KUKA KRL program: MyProgram_074().src

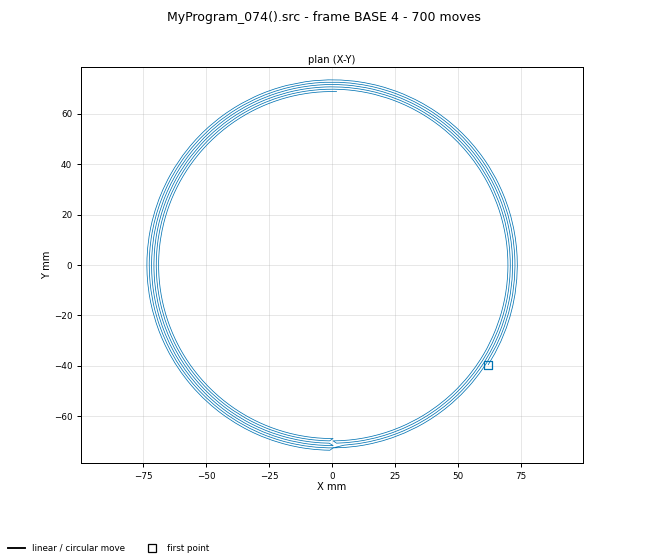
[picture p0: tool path of MyProgram_074().src in frame BASE 4, 700 of 700 moves have a stored position in this frame; points joined in program order, loops and branches not executed]
&ACCESS RVP
&REL 1
&PARAM TEMPLATE = C:\KRC\Roboter\Template\vorgabe
&PARAM EDITMASK = *
DEF MyProgram_074()
; ---- Setting reference (Base) ----
$BASE = BASE_DATA[4]

; --------------------------
; ---- Setting tool (TCP) ----
$TOOL = TOOL_DATA[3]
; --------------------------

$VEL.CP = VEL_APROX_PRINT
Startdeposition()
$VEL.CP = VEL_PRINT
LIN {X 62.0149,Y -39.5352,Z 78,A -36.8264,B 24.9007,C -2.3005,E1 25.1365,E2 121.1791} C_DIS
LIN {X 64.5776,Y -35.1935,Z 78,A -33.5799,B 24.9015,C -2.2916,E1 25.141,E2 117.9704} C_DIS
LIN {X 67.0266,Y -30.2699,Z 78,A -29.6894,B 24.9014,C -2.2926,E1 25.1458,E2 114.0982} C_DIS
LIN {X 69.1793,Y -24.9624,Z 78,A -24.6932,B 24.8988,C -2.3219,E1 25.151,E2 109.0606} C_DIS
LIN {X 70.6037,Y -20.5927,Z 78,A -21.3241,B 24.8984,C -2.3267,E1 25.1538,E2 105.6993} C_DIS
LIN {X 71.7542,Y -16.1353,Z 78,A -17.1231,B 24.8958,C -2.3562,E1 25.1566,E2 101.4529} C_DIS
LIN {X 72.6519,Y -11.4261,Z 78,A -13.91,B 24.8962,C -2.3525,E1 25.1581,E2 98.2674} C_DIS
LIN {X 73.337,Y -5.5339,Z 78,A -9.6921,B 24.8959,C -2.3552,E1 25.1594,E2 94.0681} C_DIS
LIN {X 73.5444,Y -0.3114,Z 78,A -5.4364,B 24.8943,C -2.3735,E1 25.1598,E2 89.7944} C_DIS
LIN {X 73.4622,Y 3.4708,Z 78,A -2.3202,B 24.893,C -2.3879,E1 25.1595,E2 86.6628} C_DIS
LIN {X 73.24,Y 6.6845,Z 78,A 0.445,B 24.8916,C -2.4034,E1 25.1589,E2 83.8775} C_DIS
LIN {X 72.7679,Y 10.6663,Z 78,A 3.6105,B 24.8906,C -2.4143,E1 25.1577,E2 80.7048} C_DIS
LIN {X 72.0794,Y 14.6088,Z 78,A 6.5507,B 24.8902,C -2.4187,E1 25.1561,E2 77.7715} C_DIS
LIN {X 70.9838,Y 19.2388,Z 78,A 9.4181,B 24.8914,C -2.4052,E1 25.1543,E2 74.9524} C_DIS
LIN {X 69.9868,Y 22.5982,Z 78,A 13.0379,B 24.8883,C -2.4394,E1 25.1513,E2 71.2724} C_DIS
LIN {X 68.5839,Y 26.5557,Z 78,A 15.7831,B 24.8889,C -2.4335,E1 25.1486,E2 68.5566} C_DIS
LIN {X 67.3749,Y 29.4866,Z 78,A 19.0656,B 24.886,C -2.4644,E1 25.145,E2 65.2191} C_DIS
LIN {X 65.998,Y 32.4522,Z 78,A 20.5878,B 24.8881,C -2.4414,E1 25.1432,E2 63.7593} C_DIS
LIN {X 64.9381,Y 34.5246,Z 78,A 22.9314,B 24.8863,C -2.4618,E1 25.1401,E2 61.38} C_DIS
LIN {X 62.4288,Y 38.8777,Z 78,A 26.5828,B 24.886,C -2.4644,E1 25.135,E2 57.7411} C_DIS
LIN {X 61.0309,Y 41.038,Z 78,A 29.3198,B 24.8836,C -2.4907,E1 25.1306,E2 54.9554} C_DIS
LIN {X 59.0987,Y 43.7747,Z 78,A 31.7272,B 24.8836,C -2.4912,E1 25.1266,E2 52.5586} C_DIS
LIN {X 56.5702,Y 46.9962,Z 78,A 34.4398,B 24.8841,C -2.4849,E1 25.1219,E2 49.8734} C_DIS
LIN {X 54.0669,Y 49.8561,Z 78,A 37.654,B 24.8828,C -2.4987,E1 25.1159,E2 46.6408} C_DIS
LIN {X 51.7673,Y 52.2397,Z 78,A 39.8636,B 24.8833,C -2.4936,E1 25.1116,E2 44.4527} C_DIS
LIN {X 49.0295,Y 54.8173,Z 78,A 43.1232,B 24.8819,C -2.5088,E1 25.1048,E2 41.1703} C_DIS
LIN {X 46.0603,Y 57.3357,Z 78,A 45.6068,B 24.8828,C -2.499,E1 25.0996,E2 38.7194} C_DIS
LIN {X 42.3941,Y 60.0976,Z 78,A 49.5839,B 24.8811,C -2.5164,E1 25.0906,E2 34.7154} C_DIS
LIN {X 39.5989,Y 61.974,Z 78,A 52.4619,B 24.8801,C -2.5276,E1 25.0838,E2 31.8202} C_DIS
LIN {X 35.9228,Y 64.1746,Z 78,A 55.5006,B 24.8804,C -2.524,E1 25.0765,E2 28.7992} C_DIS
LIN {X 32.8974,Y 65.7773,Z 78,A 58.0417,B 24.8804,C -2.524,E1 25.0702,E2 26.2653} C_DIS
LIN {X 28.2288,Y 67.9124,Z 78,A 62.274,B 24.8794,C -2.5347,E1 25.0594,E2 22.0179} C_DIS
LIN {X 25.5373,Y 68.9696,Z 78,A 64.6555,B 24.8789,C -2.5403,E1 25.0531,E2 19.6282} C_DIS
LIN {X 20.7617,Y 70.5536,Z 78,A 68.6434,B 24.8784,C -2.5451,E1 25.0425,E2 15.6362} C_DIS
LIN {X 17.3304,Y 71.4737,Z 78,A 71.462,B 24.8781,C -2.548,E1 25.0348,E2 12.8146} C_DIS
LIN {X 12.8619,Y 72.4115,Z 78,A 75.4013,B 24.877,C -2.5596,E1 25.0239,E2 8.8522} C_DIS
LIN {X 8.9262,Y 73.002,Z 78,A 77.3268,B 24.8799,C -2.5292,E1 25.0188,E2 7.0007} C_DIS
LIN {X 3.4859,Y 73.4628,Z 78,A 82.4313,B 24.8778,C -2.5516,E1 25.0045,E2 1.8454} C_DIS
LIN {X -1.5466,Y 73.5287,Z 78,A 86.1691,B 24.8783,C -2.5459,E1 24.9941,E2 -1.8791} C_DIS
LIN {X -7.4487,Y 73.1668,Z 78,A 91.0301,B 24.8779,C -2.5504,E1 24.9805,E2 -6.7528} C_DIS
LIN {X -10.6837,Y 72.7654,Z 78,A 93.4689,B 24.8783,C -2.5462,E1 24.9738,E2 -9.1836} C_DIS
LIN {X -17.9304,Y 71.3266,Z 78,A 98.5002,B 24.8805,C -2.5229,E1 24.9602,E2 -14.1655} C_DIS
LIN {X -19.7523,Y 70.8433,Z 78,A 100.539,B 24.8793,C -2.5356,E1 24.9546,E2 -16.238} C_DIS
LIN {X -22.8143,Y 69.9169,Z 78,A 103.3619,B 24.8788,C -2.5411,E1 24.9471,E2 -19.0788} C_DIS
LIN {X -25.9829,Y 68.802,Z 78,A 105.0367,B 24.8813,C -2.5143,E1 24.9428,E2 -20.6933} C_DIS
LIN {X -28.9327,Y 67.6153,Z 78,A 107.5191,B 24.8817,C -2.511,E1 24.9364,E2 -23.1734} C_DIS
LIN {X -30.8582,Y 66.758,Z 78,A 109.859,B 24.8803,C -2.5257,E1 24.9304,E2 -25.5541} C_DIS
LIN {X -35.9812,Y 64.142,Z 78,A 113.8595,B 24.8821,C -2.5064,E1 24.9206,E2 -29.5198} C_DIS
LIN {X -38.9619,Y 62.3763,Z 78,A 116.7798,B 24.8821,C -2.5069,E1 24.9136,E2 -32.4504} C_DIS
LIN {X -42.2245,Y 60.2162,Z 78,A 120.0318,B 24.8821,C -2.5059,E1 24.9061,E2 -35.7108} C_DIS
LIN {X -44.9358,Y 58.2203,Z 78,A 122.322,B 24.8834,C -2.4925,E1 24.901,E2 -37.9773} C_DIS
LIN {X -48.9728,Y 54.868,Z 78,A 127.1321,B 24.8826,C -2.5007,E1 24.8908,E2 -42.8257} C_DIS
LIN {X -51.4287,Y 52.5733,Z 78,A 129.2512,B 24.8843,C -2.4826,E1 24.8866,E2 -44.9105} C_DIS
LIN {X -54.0846,Y 49.8368,Z 78,A 132.8002,B 24.8837,C -2.4891,E1 24.8798,E2 -48.4904} C_DIS
LIN {X -56.3937,Y 47.2085,Z 78,A 135.9816,B 24.8833,C -2.493,E1 24.874,E2 -51.6958} C_DIS
LIN {X -59.2678,Y 43.5445,Z 78,A 138.2236,B 24.8873,C -2.4506,E1 24.8704,E2 -53.8474} C_DIS
LIN {X -62.5156,Y 38.7388,Z 78,A 142.4263,B 24.8891,C -2.4308,E1 24.8639,E2 -58.0238} C_DIS
LIN {X -64.2155,Y 35.8496,Z 78,A 145.4875,B 24.8888,C -2.4337,E1 24.8596,E2 -61.1079} C_DIS
LIN {X -65.2844,Y 33.867,Z 78,A 147.6608,B 24.8884,C -2.4383,E1 24.8567,E2 -63.3037} C_DIS
LIN {X -67.216,Y 29.8477,Z 78,A 150.7781,B 24.8901,C -2.4198,E1 24.8531,E2 -66.3937} C_DIS
LIN {X -68.7386,Y 26.1504,Z 78,A 154.2674,B 24.8901,C -2.419,E1 24.8495,E2 -69.9007} C_DIS
LIN {X -70.2736,Y 21.6899,Z 78,A 157.5058,B 24.8921,C -2.3977,E1 24.8466,E2 -73.1066} C_DIS
LIN {X -71.416,Y 17.5671,Z 78,A 160.9656,B 24.8928,C -2.3902,E1 24.8441,E2 -76.5686} C_DIS
LIN {X -72.0851,Y 14.5798,Z 78,A 163.5914,B 24.893,C -2.3882,E1 24.8426,E2 -79.2052} C_DIS
LIN {X -72.6593,Y 11.3786,Z 78,A 167.1865,B 24.8915,C -2.4048,E1 24.841,E2 -82.8613} C_DIS
LIN {X -73.2264,Y 6.8359,Z 78,A 169.709,B 24.8947,C -2.3692,E1 24.8403,E2 -85.314} C_DIS
LIN {X -73.4955,Y 2.7241,Z 78,A 172.9366,B 24.8955,C -2.3594,E1 24.8398,E2 -88.5374} C_DIS
LIN {X -73.5433,Y -0.4685,Z 78,A 176.0317,B 24.895,C -2.3656,E1 24.8398,E2 -91.6659} C_DIS
LIN {X -73.4495,Y -3.7539,Z 78,A 178.0186,B 24.8969,C -2.3442,E1 24.8401,E2 -93.6137} C_DIS
LIN {X -73.185,Y -7.2754,Z 78,A -179.5399,B 24.8983,C -2.3284,E1 24.8407,E2 -96.0323} C_DIS
LIN {X -72.628,Y -11.5765,Z 78,A -175.831,B 24.8985,C -2.3255,E1 24.8421,E2 -99.7563} C_DIS
LIN {X -72.0901,Y -14.5557,Z 78,A -173.34,B 24.8989,C -2.3213,E1 24.8434,E2 -102.252} C_DIS
LIN {X -71.3296,Y -17.9187,Z 78,A -170.224,B 24.8987,C -2.3232,E1 24.8455,E2 -105.3907} C_DIS
LIN {X -69.8642,Y -22.977,Z 78,A -166.6369,B 24.9008,C -2.2989,E1 24.8484,E2 -108.9406} C_DIS
LIN {X -68.6959,Y -26.2625,Z 78,A -163.9305,B 24.9015,C -2.2908,E1 24.851,E2 -111.6429} C_DIS
LIN {X -67.5462,Y -29.0931,Z 78,A -161.4211,B 24.9019,C -2.2871,E1 24.8537,E2 -114.1572} C_DIS
LIN {X -66.2626,Y -31.9076,Z 78,A -159.1939,B 24.9028,C -2.2761,E1 24.8563,E2 -116.3703} C_DIS
LIN {X -64.5816,Y -35.1861,Z 78,A -155.7371,B 24.9023,C -2.2822,E1 24.8609,E2 -119.8601} C_DIS
LIN {X -62.3685,Y -38.9743,Z 78,A -152.1844,B 24.9028,C -2.2765,E1 24.8661,E2 -123.4176} C_DIS
LIN {X -59.9501,Y -42.6008,Z 78,A -148.9097,B 24.9037,C -2.2652,E1 24.8713,E2 -126.6813} C_DIS
LIN {X -57.585,Y -45.7474,Z 78,A -146.2138,B 24.9051,C -2.249,E1 24.8759,E2 -129.3513} C_DIS
LIN {X -55.9426,Y -47.7416,Z 78,A -144.1882,B 24.9055,C -2.2447,E1 24.8795,E2 -131.376} C_DIS
LIN {X -54.4689,Y -49.4179,Z 78,A -142.4514,B 24.9058,C -2.2408,E1 24.8828,E2 -133.1111} C_DIS
LIN {X -51.2843,Y -52.7143,Z 78,A -138.5837,B 24.9058,C -2.2405,E1 24.8904,E2 -136.9947} C_DIS
LIN {X -47.9483,Y -55.7664,Z 78,A -135.6851,B 24.9077,C -2.2184,E1 24.8963,E2 -139.8522} C_DIS
LIN {X -44.9917,Y -58.1772,Z 78,A -132.2305,B 24.9071,C -2.2249,E1 24.9039,E2 -143.335} C_DIS
LIN {X -42.2829,Y -60.1758,Z 78,A -129.3799,B 24.9071,C -2.2262,E1 24.9104,E2 -146.1986} C_DIS
LIN {X -38.3696,Y -62.7427,Z 78,A -125.7958,B 24.9076,C -2.2191,E1 24.9189,E2 -149.7773} C_DIS
LIN {X -34.6931,Y -64.849,Z 78,A -121.9218,B 24.9068,C -2.2293,E1 24.9285,E2 -153.6865} C_DIS
LIN {X -31.2662,Y -66.5681,Z 78,A -119.5584,B 24.9084,C -2.2099,E1 24.9343,E2 -156.0098} C_DIS
LIN {X -28.0543,Y -67.9846,Z 78,A -116.8143,B 24.9086,C -2.2073,E1 24.9414,E2 -158.7541} C_DIS
LIN {X -23.7093,Y -69.6185,Z 78,A -112.9079,B 24.9082,C -2.2117,E1 24.9517,E2 -162.6787} C_DIS
LIN {X -19.5219,Y -70.9064,Z 78,A -109.3766,B 24.9082,C -2.2126,E1 24.9612,E2 -166.2177} C_DIS
LIN {X -16.3801,Y -71.6976,Z 78,A -107.7838,B 24.9103,C -2.187,E1 24.9654,E2 -167.7519} C_DIS
LIN {X -12.9712,Y -72.3918,Z 78,A -105.3498,B 24.911,C -2.1788,E1 24.972,E2 -170.169} C_DIS
LIN {X -10.941,Y -72.727,Z 78,A -102.2703,B 24.9078,C -2.2172,E1 24.9808,E2 -173.3425} C_DIS
LIN {X -7.0298,Y -73.2084,Z 78,A -100.245,B 24.9101,C -2.1891,E1 24.9862,E2 -175.3022} C_DIS
LIN {X -3.0309,Y -73.4824,Z 78,A -97.4489,B 24.9108,C -2.1806,E1 24.994,E2 -178.079} C_DIS
LIN {X -0.903,Y -73.5406,Z 78,A -94.0962,B 24.907,C -2.2264,E1 25.0036,E2 -181.5406} C_DIS
LIN {X -0.903,Y -73.5406,Z 78,A -94.0962,B 24.907,C -2.2264,E1 25.0036,E2 -181.5406} C_DIS
Enddeposition()
LIN {X 0.4401,Y -72.5902,Z 78,A -93.7193,B 24.9072,C -2.2247,E1 25.0047,E2 -181.9133} C_DIS
Startdeposition()
$VEL.CP = VEL_PRINT
LIN {X -1.5403,Y -72.5975,Z 78,A -97.2134,B 24.9114,C -2.1733,E1 24.9946,E2 -178.2974} C_DIS
LIN {X -6.3605,Y -72.3352,Z 78,A -102.0186,B 24.9134,C -2.1483,E1 24.981,E2 -173.4305} C_DIS
LIN {X -11.1322,Y -71.7552,Z 78,A -104.0226,B 24.9097,C -2.1942,E1 24.9758,E2 -171.5341} C_DIS
LIN {X -15.5858,Y -70.9213,Z 78,A -107.7338,B 24.9099,C -2.192,E1 24.9656,E2 -167.8137} C_DIS
LIN {X -19.0944,Y -70.0583,Z 78,A -111.0187,B 24.9106,C -2.1826,E1 24.9566,E2 -164.5018} C_DIS
LIN {X -21.8748,Y -69.2399,Z 78,A -113.5308,B 24.911,C -2.1787,E1 24.9498,E2 -161.9761} C_DIS
LIN {X -25.901,Y -67.8374,Z 78,A -116.8325,B 24.9106,C -2.1832,E1 24.9412,E2 -158.6783} C_DIS
LIN {X -28.4017,Y -66.8291,Z 78,A -119.2336,B 24.911,C -2.1787,E1 24.935,E2 -156.261} C_DIS
LIN {X -32.57,Y -64.8993,Z 78,A -122.8507,B 24.9106,C -2.1831,E1 24.9259,E2 -152.6452} C_DIS
LIN {X -37.5446,Y -62.1544,Z 78,A -127.452,B 24.9103,C -2.1865,E1 24.9147,E2 -148.0383} C_DIS
LIN {X -41.535,Y -59.5616,Z 78,A -130.5191,B 24.9085,C -2.2089,E1 24.9077,E2 -145.0143} C_DIS
LIN {X -44.3548,Y -57.4925,Z 78,A -133.5609,B 24.9086,C -2.2069,E1 24.9009,E2 -141.957} C_DIS
LIN {X -46.925,Y -55.415,Z 78,A -135.6957,B 24.9073,C -2.2229,E1 24.8963,E2 -139.8522} C_DIS
LIN {X -50.093,Y -52.5699,Z 78,A -140.3066,B 24.9092,C -2.2003,E1 24.8867,E2 -135.1687} C_DIS
LIN {X -52.715,Y -49.9393,Z 78,A -142.4082,B 24.9071,C -2.2258,E1 24.8828,E2 -133.1187} C_DIS
LIN {X -55.1223,Y -47.2686,Z 78,A -145.38,B 24.9068,C -2.229,E1 24.8773,E2 -130.1412} C_DIS
LIN {X -57.2915,Y -44.6156,Z 78,A -147.6991,B 24.9055,C -2.2442,E1 24.8733,E2 -127.8475} C_DIS
LIN {X -59.5737,Y -41.5176,Z 78,A -150.8597,B 24.9051,C -2.2487,E1 24.8681,E2 -124.6824} C_DIS
LIN {X -61.8421,Y -38.0586,Z 78,A -154.1792,B 24.9045,C -2.2557,E1 24.863,E2 -121.3629} C_DIS
LIN {X -63.9816,Y -34.3371,Z 78,A -157.9635,B 24.9045,C -2.2557,E1 24.8578,E2 -117.5587} C_DIS
LIN {X -65.6101,Y -31.1157,Z 78,A -161.4614,B 24.9051,C -2.2491,E1 24.8536,E2 -114.026} C_DIS
LIN {X -67.1485,Y -27.6387,Z 78,A -164.6161,B 24.9047,C -2.2542,E1 24.8502,E2 -110.866} C_DIS
LIN {X -68.6294,Y -23.7246,Z 78,A -166.7374,B 24.9016,C -2.2901,E1 24.8483,E2 -108.8184} C_DIS
LIN {X -69.2974,Y -21.6921,Z 78,A -169.606,B 24.9034,C -2.2689,E1 24.8459,E2 -105.8827} C_DIS
LIN {X -70.4208,Y -17.714,Z 78,A -171.9981,B 24.9009,C -2.2979,E1 24.8442,E2 -103.5458} C_DIS
LIN {X -70.9767,Y -15.3319,Z 78,A -174.239,B 24.901,C -2.2969,E1 24.8429,E2 -101.2895} C_DIS
LIN {X -71.9087,Y -10.0935,Z 78,A -178.0344,B 24.8991,C -2.3188,E1 24.8412,E2 -97.5238} C_DIS
LIN {X -72.2407,Y -7.352,Z 78,A 179.9213,B 24.8983,C -2.3286,E1 24.8405,E2 -95.4907} C_DIS
LIN {X -72.5297,Y -3.511,Z 78,A 176.2296,B 24.8987,C -2.3238,E1 24.8399,E2 -91.7652} C_DIS
LIN {X -72.611,Y 0.6577,Z 78,A 173.3066,B 24.8971,C -2.3423,E1 24.8399,E2 -88.8689} C_DIS
LIN {X -72.5207,Y 3.6858,Z 78,A 171.2509,B 24.8957,C -2.3573,E1 24.84,E2 -86.8366} C_DIS
LIN {X -72.2735,Y 7.0282,Z 78,A 167.488,B 24.8972,C -2.3411,E1 24.841,E2 -83.0126} C_DIS
LIN {X -71.8395,Y 10.581,Z 78,A 165.357,B 24.895,C -2.3652,E1 24.8418,E2 -80.9264} C_DIS
LIN {X -71.4317,Y 13.0495,Z 78,A 162.9633,B 24.8953,C -2.3623,E1 24.843,E2 -78.5114} C_DIS
LIN {X -70.7012,Y 16.5566,Z 78,A 159.5591,B 24.8956,C -2.3586,E1 24.8452,E2 -75.0784} C_DIS
LIN {X -69.6173,Y 20.6438,Z 78,A 157.5721,B 24.892,C -2.3985,E1 24.8466,E2 -73.1753} C_DIS
LIN {X -68.4133,Y 24.3394,Z 78,A 153.7756,B 24.8926,C -2.3918,E1 24.85,E2 -69.3411} C_DIS
LIN {X -66.9712,Y 28.0645,Z 78,A 151.1206,B 24.8908,C -2.4123,E1 24.8527,E2 -66.7202} C_DIS
LIN {X -65.3212,Y 31.7169,Z 78,A 147.7001,B 24.8905,C -2.4159,E1 24.8568,E2 -63.2896} C_DIS
LIN {X -63.8021,Y 34.6702,Z 78,A 145.108,B 24.8897,C -2.4241,E1 24.8601,E2 -60.7035} C_DIS
LIN {X -61.8525,Y 38.0413,Z 78,A 141.0659,B 24.8909,C -2.4113,E1 24.866,E2 -56.61} C_DIS
LIN {X -59.6134,Y 41.4605,Z 78,A 138.9818,B 24.8878,C -2.4455,E1 24.8692,E2 -54.5972} C_DIS
LIN {X -58.5543,Y 42.9433,Z 78,A 136.1975,B 24.8902,C -2.4194,E1 24.874,E2 -51.737} C_DIS
LIN {X -55.7144,Y 46.5691,Z 78,A 133.3525,B 24.8877,C -2.4462,E1 24.8789,E2 -48.943} C_DIS
LIN {X -52.5449,Y 50.1189,Z 78,A 129.9963,B 24.886,C -2.4645,E1 24.8852,E2 -45.6157} C_DIS
LIN {X -48.35,Y 54.1759,Z 78,A 124.8913,B 24.886,C -2.4638,E1 24.8956,E2 -40.488} C_DIS
LIN {X -44.2936,Y 57.5396,Z 78,A 120.5645,B 24.8856,C -2.4689,E1 24.9051,E2 -36.1572} C_DIS
LIN {X -39.9033,Y 60.6668,Z 78,A 116.8787,B 24.8836,C -2.4903,E1 24.9134,E2 -32.51} C_DIS
LIN {X -37.3511,Y 62.2709,Z 78,A 114.5657,B 24.883,C -2.4962,E1 24.9189,E2 -30.2037} C_DIS
LIN {X -35.3335,Y 63.4373,Z 78,A 112.286,B 24.8837,C -2.4891,E1 24.9245,E2 -27.9004} C_DIS
LIN {X -30.6059,Y 65.8484,Z 78,A 108.9963,B 24.8811,C -2.517,E1 24.9326,E2 -24.6684} C_DIS
LIN {X -26.6576,Y 67.5434,Z 78,A 105.0286,B 24.8819,C -2.5079,E1 24.9429,E2 -20.6701} C_DIS
LIN {X -22.7333,Y 68.9644,Z 78,A 101.938,B 24.8811,C -2.5169,E1 24.951,E2 -17.5947} C_DIS
LIN {X -18.8094,Y 70.1353,Z 78,A 98.6328,B 24.8809,C -2.5185,E1 24.9599,E2 -14.288} C_DIS
LIN {X -14.7924,Y 71.0912,Z 78,A 95.2009,B 24.8811,C -2.5172,E1 24.9692,E2 -10.8486} C_DIS
LIN {X -10.3563,Y 71.8714,Z 78,A 91.266,B 24.8817,C -2.5104,E1 24.9801,E2 -6.8938} C_DIS
LIN {X -6.6457,Y 72.3088,Z 78,A 87.8411,B 24.8827,C -2.5002,E1 24.9897,E2 -3.4429} C_DIS
LIN {X -2.8742,Y 72.5571,Z 78,A 85.6748,B 24.8807,C -2.5214,E1 24.9956,E2 -1.3264} C_DIS
LIN {X 2.7685,Y 72.5613,Z 78,A 81.5646,B 24.8798,C -2.5307,E1 25.007,E2 2.7613} C_DIS
LIN {X 7.1833,Y 72.2584,Z 78,A 77.8819,B 24.8803,C -2.5257,E1 25.0173,E2 6.4542} C_DIS
LIN {X 12.2744,Y 71.5691,Z 78,A 73.9452,B 24.8801,C -2.5277,E1 25.0282,E2 10.3828} C_DIS
LIN {X 15.8244,Y 70.8692,Z 78,A 70.7772,B 24.881,C -2.5183,E1 25.0369,E2 13.569} C_DIS
LIN {X 18.9884,Y 70.0869,Z 78,A 68.0915,B 24.8814,C -2.5138,E1 25.0441,E2 16.2612} C_DIS
LIN {X 22.9158,Y 68.9035,Z 78,A 64.8524,B 24.8816,C -2.5113,E1 25.0528,E2 19.5004} C_DIS
LIN {X 25.3422,Y 68.049,Z 78,A 62.5806,B 24.8824,C -2.5031,E1 25.0588,E2 21.7868} C_DIS
LIN {X 29.5259,Y 66.3391,Z 78,A 59.0606,B 24.8826,C -2.5005,E1 25.0678,E2 25.3046} C_DIS
LIN {X 32.6326,Y 64.8693,Z 78,A 56.3222,B 24.883,C -2.4964,E1 25.0746,E2 28.0453} C_DIS
LIN {X 37.1431,Y 62.3953,Z 78,A 52.5098,B 24.883,C -2.4973,E1 25.0839,E2 31.8441} C_DIS
LIN {X 39.8844,Y 60.6793,Z 78,A 49.8553,B 24.8836,C -2.4906,E1 25.0901,E2 34.5059} C_DIS
LIN {X 43.8644,Y 57.8683,Z 78,A 46.2697,B 24.8836,C -2.4911,E1 25.0982,E2 38.0778} C_DIS
LIN {X 46.424,Y 55.8349,Z 78,A 43.4145,B 24.8847,C -2.4788,E1 25.1044,E2 40.9511} C_DIS
LIN {X 49.9897,Y 52.6671,Z 78,A 40.0556,B 24.8843,C -2.4824,E1 25.1113,E2 44.288} C_DIS
LIN {X 52.0972,Y 50.5834,Z 78,A 36.7563,B 24.8872,C -2.4511,E1 25.1178,E2 47.6472} C_DIS
LIN {X 54.8193,Y 47.6195,Z 78,A 34.4891,B 24.8856,C -2.4689,E1 25.1219,E2 49.8621} C_DIS
LIN {X 56.7747,Y 45.271,Z 78,A 31.6954,B 24.8871,C -2.4527,E1 25.1269,E2 52.6812} C_DIS
LIN {X 59.7464,Y 41.2692,Z 78,A 28.2101,B 24.8868,C -2.4555,E1 25.1325,E2 56.143} C_DIS
LIN {X 61.4607,Y 38.67,Z 78,A 24.6138,B 24.8903,C -2.4175,E1 25.138,E2 59.811} C_DIS
LIN {X 63.8046,Y 34.6657,Z 78,A 22.0991,B 24.8883,C -2.4397,E1 25.1413,E2 62.2601} C_DIS
LIN {X 65.6837,Y 30.9582,Z 78,A 18.7462,B 24.8893,C -2.4286,E1 25.1454,E2 65.6214} C_DIS
LIN {X 67.5155,Y 26.7288,Z 78,A 15.5727,B 24.8891,C -2.4314,E1 25.1489,E2 68.7709} C_DIS
LIN {X 68.2892,Y 24.6853,Z 78,A 13.2462,B 24.8911,C -2.4092,E1 25.1511,E2 71.1367} C_DIS
LIN {X 69.7825,Y 20.0803,Z 78,A 9.7819,B 24.8911,C -2.408,E1 25.154,E2 74.5842} C_DIS
LIN {X 71.1056,Y 14.722,Z 78,A 5.4941,B 24.8922,C -2.3967,E1 25.1568,E2 78.8739} C_DIS
LIN {X 71.9388,Y 9.8818,Z 78,A 1.0849,B 24.8947,C -2.3694,E1 25.1587,E2 83.3217} C_DIS
LIN {X 72.4268,Y 5.2153,Z 78,A -2.0955,B 24.8944,C -2.3727,E1 25.1595,E2 86.4755} C_DIS
LIN {X 72.5861,Y 2.009,Z 78,A -4.6685,B 24.8952,C -2.3635,E1 25.1598,E2 89.0548} C_DIS
LIN {X 72.6114,Y -0.594,Z 78,A -6.9772,B 24.8964,C -2.3497,E1 25.1598,E2 91.3824} C_DIS
LIN {X 72.4059,Y -5.4963,Z 78,A -11.0013,B 24.8979,C -2.333,E1 25.1591,E2 95.4219} C_DIS
LIN {X 71.7497,Y -11.1679,Z 78,A -14.7551,B 24.8972,C -2.3403,E1 25.1577,E2 99.1365} C_DIS
LIN {X 71.4279,Y -13.0697,Z 78,A -17.0569,B 24.8996,C -2.3131,E1 25.1566,E2 101.489} C_DIS
LIN {X 70.1423,Y -18.7835,Z 78,A -21.0411,B 24.8993,C -2.3168,E1 25.154,E2 105.4413} C_DIS
LIN {X 68.4563,Y -24.2177,Z 78,A -25.2646,B 24.8998,C -2.3106,E1 25.1504,E2 109.6555} C_DIS
LIN {X 67.1016,Y -27.7519,Z 78,A -28.6725,B 24.9017,C -2.2894,E1 25.1469,E2 113.0946} C_DIS
LIN {X 65.1265,Y -32.1138,Z 78,A -32.6589,B 24.9031,C -2.2723,E1 25.1421,E2 117.1} C_DIS
LIN {X 61.5029,Y -38.6025,Z 78,A -37.7524,B 24.9027,C -2.2775,E1 25.1351,E2 122.1548} C_DIS
LIN {X 59.8419,Y -41.1303,Z 78,A -40.4332,B 24.904,C -2.2625,E1 25.1309,E2 124.8577} C_DIS
LIN {X 58.2027,Y -43.4193,Z 78,A -42.8532,B 24.905,C -2.2509,E1 25.1269,E2 127.2935} C_DIS
LIN {X 55.5723,Y -46.7395,Z 78,A -45.8602,B 24.9049,C -2.2516,E1 25.1216,E2 130.2848} C_DIS
LIN {X 54.2613,Y -48.2546,Z 78,A -47.9078,B 24.9063,C -2.2345,E1 25.1178,E2 132.3638} C_DIS
LIN {X 51.1951,Y -51.4961,Z 78,A -51.2602,B 24.9067,C -2.2306,E1 25.1113,E2 135.7108} C_DIS
LIN {X 47.6851,Y -54.762,Z 78,A -54.8564,B 24.907,C -2.2271,E1 25.1038,E2 139.3009} C_DIS
LIN {X 44.6981,Y -57.2264,Z 78,A -58.062,B 24.9079,C -2.2163,E1 25.0968,E2 142.52} C_DIS
LIN {X 41.9624,Y -59.2618,Z 78,A -60.5827,B 24.9079,C -2.2155,E1 25.0912,E2 145.0336} C_DIS
LIN {X 39.158,Y -61.1506,Z 78,A -62.9782,B 24.9077,C -2.2179,E1 25.0856,E2 147.4156} C_DIS
LIN {X 36.3366,Y -62.8683,Z 78,A -66.0755,B 24.9092,C -2.1996,E1 25.0781,E2 150.5466} C_DIS
LIN {X 33.766,Y -64.2853,Z 78,A -68.5201,B 24.9099,C -2.1922,E1 25.072,E2 153.0018} C_DIS
LIN {X 28.7007,Y -66.7017,Z 78,A -72.6086,B 24.9097,C -2.1946,E1 25.0617,E2 157.0743} C_DIS
LIN {X 23.8439,Y -68.5875,Z 78,A -76.9358,B 24.9106,C -2.1834,E1 25.0503,E2 161.419} C_DIS
LIN {X 20.0624,Y -69.7876,Z 78,A -79.3866,B 24.9094,C -2.198,E1 25.0439,E2 163.8307} C_DIS
LIN {X 15.8946,Y -70.8531,Z 78,A -82.834,B 24.9098,C -2.1932,E1 25.0346,E2 167.2843} C_DIS
LIN {X 12.6894,Y -71.4964,Z 78,A -85.9596,B 24.9111,C -2.1766,E1 25.0259,E2 170.4457} C_DIS
LIN {X 9.7952,Y -71.9511,Z 78,A -88.3417,B 24.9114,C -2.1732,E1 25.0193,E2 172.8339} C_DIS
LIN {X 5.0583,Y -72.4374,Z 78,A -91.4313,B 24.9101,C -2.1887,E1 25.0108,E2 175.8847} C_DIS
LIN {X 0.4401,Y -72.5902,Z 78,A -93.7169,B 24.9072,C -2.2237,E1 25.0047,E2 178.0866} C_DIS
Enddeposition()
LIN {X 0.4401,Y -72.5902,Z 78,A -93.7169,B 24.9072,C -2.2237,E1 25.0047,E2 178.0866} C_DIS
Startdeposition()
$VEL.CP = VEL_PRINT
LIN {X 4.7456,Y -71.5252,Z 78,A -90.38,B 24.9061,C -2.2377,E1 25.014,E2 174.7179} C_DIS
LIN {X 10.2822,Y -70.9414,Z 78,A -86.6436,B 24.9074,C -2.2214,E1 25.0243,E2 171.0228} C_DIS
LIN {X 14.8753,Y -70.1232,Z 78,A -82.6289,B 24.9065,C -2.232,E1 25.0354,E2 166.9876} C_DIS
LIN {X 19.1531,Y -69.0775,Z 78,A -79.4537,B 24.907,C -2.2263,E1 25.0439,E2 163.8307} C_DIS
LIN {X 22.1838,Y -68.1635,Z 78,A -76.5584,B 24.9059,C -2.2391,E1 25.0517,E2 160.9103} C_DIS
LIN {X 25.58,Y -66.9633,Z 78,A -73.669,B 24.9056,C -2.2432,E1 25.0593,E2 158.0173} C_DIS
LIN {X 28.1777,Y -65.913,Z 78,A -70.7706,B 24.9038,C -2.2645,E1 25.0668,E2 155.0752} C_DIS
LIN {X 31.4442,Y -64.4179,Z 78,A -68.6285,B 24.9051,C -2.2489,E1 25.0721,E2 152.9757} C_DIS
LIN {X 34.006,Y -63.1031,Z 78,A -65.4024,B 24.9026,C -2.2786,E1 25.0802,E2 149.6887} C_DIS
LIN {X 37.6579,Y -60.9951,Z 78,A -63.3344,B 24.9052,C -2.2484,E1 25.085,E2 147.6984} C_DIS
LIN {X 40.9313,Y -58.8473,Z 78,A -59.8082,B 24.9037,C -2.2656,E1 25.0932,E2 144.1434} C_DIS
LIN {X 44.6413,Y -56.0849,Z 78,A -55.918,B 24.9026,C -2.2788,E1 25.1018,E2 140.2362} C_DIS
LIN {X 46.9592,Y -54.1597,Z 78,A -53.8364,B 24.9029,C -2.275,E1 25.1062,E2 138.1717} C_DIS
LIN {X 49.4403,Y -51.9046,Z 78,A -51.189,B 24.9024,C -2.2803,E1 25.1116,E2 135.5226} C_DIS
LIN {X 51.6215,Y -49.7352,Z 78,A -48.6933,B 24.9018,C -2.2873,E1 25.1165,E2 133.0209} C_DIS
LIN {X 54.1776,Y -46.9387,Z 78,A -45.9867,B 24.902,C -2.2858,E1 25.1216,E2 130.33} C_DIS
LIN {X 55.8769,Y -44.9022,Z 78,A -43.2005,B 24.8999,C -2.3103,E1 25.1265,E2 127.4988} C_DIS
LIN {X 58.5293,Y -41.3847,Z 78,A -39.4132,B 24.8984,C -2.3275,E1 25.1328,E2 123.6891} C_DIS
LIN {X 60.4416,Y -38.5387,Z 78,A -37.643,B 24.9001,C -2.3072,E1 25.1354,E2 121.9756} C_DIS
LIN {X 62.7833,Y -34.5948,Z 78,A -34.0069,B 24.8993,C -2.3168,E1 25.1405,E2 118.3358} C_DIS
LIN {X 64.3772,Y -31.5262,Z 78,A -30.4988,B 24.8967,C -2.3464,E1 25.145,E2 114.7764} C_DIS
LIN {X 66.0027,Y -27.9648,Z 78,A -27.8624,B 24.8971,C -2.3415,E1 25.1479,E2 112.1659} C_DIS
LIN {X 67.4223,Y -24.3447,Z 78,A -24.9219,B 24.8967,C -2.3461,E1 25.1508,E2 109.2309} C_DIS
LIN {X 68.732,Y -20.3541,Z 78,A -21.6942,B 24.8961,C -2.3527,E1 25.1535,E2 106.0058} C_DIS
LIN {X 69.3673,Y -18.0723,Z 78,A -19.3717,B 24.8945,C -2.3711,E1 25.1552,E2 103.6533} C_DIS
LIN {X 70.2697,Y -14.1634,Z 78,A -16.1801,B 24.8936,C -2.3807,E1 25.1571,E2 100.4575} C_DIS
LIN {X 70.8276,Y -11.0375,Z 78,A -13.4231,B 24.8923,C -2.3952,E1 25.1583,E2 97.6827} C_DIS
LIN {X 71.4579,Y -5.6701,Z 78,A -10.2024,B 24.894,C -2.3771,E1 25.1593,E2 94.5237} C_DIS
LIN {X 71.6804,Y -0.5619,Z 78,A -5.9042,B 24.8923,C -2.3961,E1 25.1598,E2 90.2062} C_DIS
LIN {X 71.6628,Y 1.7243,Z 78,A -3.383,B 24.8899,C -2.4219,E1 25.1596,E2 87.639} C_DIS
LIN {X 71.4672,Y 5.5535,Z 78,A -0.6145,B 24.8899,C -2.423,E1 25.1591,E2 84.8843} C_DIS
LIN {X 71.0755,Y 9.3088,Z 78,A 2.2221,B 24.8894,C -2.4272,E1 25.1582,E2 82.0545} C_DIS
LIN {X 70.4749,Y 13.1001,Z 78,A 5.3987,B 24.8883,C -2.4398,E1 25.1568,E2 78.8668} C_DIS
LIN {X 69.846,Y 16.1216,Z 78,A 7.8978,B 24.8875,C -2.4483,E1 25.1552,E2 76.3622} C_DIS
LIN {X 69.2762,Y 18.4189,Z 78,A 9.6227,B 24.8875,C -2.4492,E1 25.154,E2 74.6451} C_DIS
LIN {X 68.5086,Y 21.0943,Z 78,A 12.6696,B 24.8846,C -2.4795,E1 25.1515,E2 71.5439} C_DIS
LIN {X 67.3709,Y 24.4855,Z 78,A 14.6422,B 24.8862,C -2.4624,E1 25.1497,E2 69.6229} C_DIS
LIN {X 66.078,Y 27.7861,Z 78,A 17.4411,B 24.8855,C -2.4695,E1 25.1468,E2 66.8227} C_DIS
LIN {X 64.7824,Y 30.6838,Z 78,A 20.3834,B 24.8838,C -2.4882,E1 25.1433,E2 63.8521} C_DIS
LIN {X 63.3875,Y 33.4724,Z 78,A 23.0827,B 24.8826,C -2.5008,E1 25.1398,E2 61.1372} C_DIS
LIN {X 60.4909,Y 38.4619,Z 78,A 27.1516,B 24.8829,C -2.4974,E1 25.134,E2 57.097} C_DIS
LIN {X 58.0066,Y 42.1153,Z 78,A 30.7393,B 24.882,C -2.5078,E1 25.1282,E2 53.5025} C_DIS
LIN {X 56.4708,Y 44.1539,Z 78,A 32.7586,B 24.8815,C -2.5121,E1 25.1248,E2 51.4826} C_DIS
LIN {X 54.3523,Y 46.7365,Z 78,A 35.3621,B 24.8811,C -2.5163,E1 25.1201,E2 48.8809} C_DIS
LIN {X 52.248,Y 49.0767,Z 78,A 38.0654,B 24.8801,C -2.5271,E1 25.115,E2 46.164} C_DIS
LIN {X 50.0307,Y 51.3367,Z 78,A 40.8868,B 24.8788,C -2.5404,E1 25.1093,E2 43.3229} C_DIS
LIN {X 46.6072,Y 54.4626,Z 78,A 44.0428,B 24.8796,C -2.5325,E1 25.1028,E2 40.1982} C_DIS
LIN {X 44.1184,Y 56.4988,Z 78,A 46.7,B 24.8789,C -2.5395,E1 25.097,E2 37.5343} C_DIS
LIN {X 41.3446,Y 58.5587,Z 78,A 49.8804,B 24.8774,C -2.5557,E1 25.0897,E2 34.3268} C_DIS
LIN {X 38.4968,Y 60.4685,Z 78,A 52.2029,B 24.8781,C -2.5485,E1 25.0843,E2 32.0288} C_DIS
LIN {X 34.7944,Y 62.6718,Z 78,A 55.9316,B 24.8769,C -2.5611,E1 25.0752,E2 28.2815} C_DIS
LIN {X 31.8195,Y 64.2331,Z 78,A 58.1051,B 24.8779,C -2.5507,E1 25.0699,E2 26.1385} C_DIS
LIN {X 27.457,Y 66.2168,Z 78,A 62.7104,B 24.8755,C -2.5755,E1 25.058,E2 21.4856} C_DIS
LIN {X 24.3786,Y 67.4099,Z 78,A 64.7509,B 24.8768,C -2.562,E1 25.0527,E2 19.4813} C_DIS
LIN {X 19.894,Y 68.8673,Z 78,A 68.8778,B 24.8756,C -2.5742,E1 25.0416,E2 15.3328} C_DIS
LIN {X 16.207,Y 69.8263,Z 78,A 71.4099,B 24.8767,C -2.5626,E1 25.0349,E2 12.8321} C_DIS
LIN {X 13.3918,Y 70.4206,Z 78,A 73.889,B 24.8762,C -2.5682,E1 25.028,E2 10.3427} C_DIS
LIN {X 8.4945,Y 71.1775,Z 78,A 77.6599,B 24.8766,C -2.5643,E1 25.0177,E2 6.5844} C_DIS
LIN {X 5.6815,Y 71.4569,Z 78,A 80.1178,B 24.876,C -2.5696,E1 25.0108,E2 4.1154} C_DIS
LIN {X 2.0734,Y 71.6526,Z 78,A 83.3877,B 24.8751,C -2.5791,E1 25.0016,E2 0.8237} C_DIS
LIN {X -2.6527,Y 71.6346,Z 78,A 86.6386,B 24.8765,C -2.5648,E1 24.9926,E2 -2.3934} C_DIS
LIN {X -5.5367,Y 71.4685,Z 78,A 89.261,B 24.8758,C -2.5716,E1 24.9853,E2 -5.0332} C_DIS
LIN {X -8.5001,Y 71.1769,Z 78,A 92.1858,B 24.8747,C -2.5839,E1 24.9771,E2 -7.9891} C_DIS
LIN {X -12.2549,Y 70.6285,Z 78,A 94.2077,B 24.8773,C -2.5567,E1 24.9717,E2 -9.9481} C_DIS
LIN {X -14.8215,Y 70.1346,Z 78,A 96.5057,B 24.877,C -2.5601,E1 24.9654,E2 -12.2569} C_DIS
LIN {X -17.8595,Y 69.422,Z 78,A 99.8666,B 24.8751,C -2.579,E1 24.9561,E2 -15.6676} C_DIS
LIN {X -21.6353,Y 68.3408,Z 78,A 101.9911,B 24.8779,C -2.5507,E1 24.9506,E2 -17.7284} C_DIS
LIN {X -24.561,Y 67.3434,Z 78,A 104.8128,B 24.8773,C -2.5561,E1 24.9431,E2 -20.5685} C_DIS
LIN {X -28.6535,Y 65.7065,Z 78,A 108.1234,B 24.8783,C -2.5461,E1 24.9347,E2 -23.8627} C_DIS
LIN {X -31.4543,Y 64.4141,Z 78,A 110.6726,B 24.8785,C -2.5443,E1 24.9282,E2 -26.4141} C_DIS
LIN {X -34.6857,Y 62.7325,Z 78,A 113.5777,B 24.879,C -2.5393,E1 24.9211,E2 -29.3155} C_DIS
LIN {X -37.5827,Y 61.0405,Z 78,A 115.996,B 24.88,C -2.5283,E1 24.9153,E2 -31.715} C_DIS
LIN {X -39.265,Y 59.9724,Z 78,A 117.9079,B 24.8796,C -2.5327,E1 24.9108,E2 -33.6436} C_DIS
LIN {X -42.1667,Y 57.9683,Z 78,A 120.7317,B 24.8801,C -2.5272,E1 24.9044,E2 -36.4641} C_DIS
LIN {X -44.6227,Y 56.1002,Z 78,A 124.0535,B 24.8787,C -2.542,E1 24.897,E2 -39.8334} C_DIS
LIN {X -47.6444,Y 53.5577,Z 78,A 125.9008,B 24.8823,C -2.5046,E1 24.8933,E2 -41.5988} C_DIS
LIN {X -50.9656,Y 50.4071,Z 78,A 129.8828,B 24.8823,C -2.5034,E1 24.8853,E2 -45.5944} C_DIS
LIN {X -55.0352,Y 45.9296,Z 78,A 135.6083,B 24.8816,C -2.5116,E1 24.8746,E2 -51.3653} C_DIS
LIN {X -57.2232,Y 43.1729,Z 78,A 137.8458,B 24.8835,C -2.491,E1 24.8709,E2 -53.5642} C_DIS
LIN {X -59.979,Y 39.2549,Z 78,A 141.8221,B 24.8842,C -2.4839,E1 24.8646,E2 -57.5432} C_DIS
LIN {X -61.8182,Y 36.289,Z 78,A 144.8547,B 24.8844,C -2.4815,E1 24.8603,E2 -60.5858} C_DIS
LIN {X -63.9731,Y 32.3399,Z 78,A 148.8046,B 24.8846,C -2.479,E1 24.8552,E2 -64.551} C_DIS
LIN {X -65.5804,Y 28.9428,Z 78,A 150.9695,B 24.8872,C -2.4512,E1 24.8528,E2 -66.6612} C_DIS
LIN {X -66.7013,Y 26.2546,Z 78,A 153.3809,B 24.8877,C -2.446,E1 24.8503,E2 -69.0738} C_DIS
LIN {X -68.5791,Y 20.8668,Z 78,A 157.6371,B 24.8896,C -2.4252,E1 24.8465,E2 -73.3045} C_DIS
LIN {X -69.6392,Y 16.9928,Z 78,A 161.01,B 24.8902,C -2.4188,E1 24.8441,E2 -76.6817} C_DIS
LIN {X -70.4464,Y 13.257,Z 78,A 164.0995,B 24.891,C -2.4099,E1 24.8423,E2 -79.7683} C_DIS
LIN {X -70.8079,Y 11.165,Z 78,A 165.8492,B 24.8914,C -2.4058,E1 24.8415,E2 -81.5183} C_DIS
LIN {X -71.3182,Y 7.221,Z 78,A 169.5456,B 24.8913,C -2.4072,E1 24.8403,E2 -85.2403} C_DIS
LIN {X -71.612,Y 3.1786,Z 78,A 172.3552,B 24.8931,C -2.3873,E1 24.8399,E2 -88.0193} C_DIS
LIN {X -71.6827,Y 0.204,Z 78,A 174.8132,B 24.8936,C -2.3815,E1 24.8398,E2 -90.4783} C_DIS
LIN {X -71.6082,Y -3.2677,Z 78,A 177.8285,B 24.8939,C -2.3781,E1 24.8401,E2 -93.5036} C_DIS
LIN {X -71.4035,Y -6.3233,Z 78,A -179.9861,B 24.8951,C -2.3646,E1 24.8406,E2 -95.6697} C_DIS
LIN {X -71.0987,Y -9.13,Z 78,A -177.7635,B 24.8958,C -2.3568,E1 24.8413,E2 -97.887} C_DIS
LIN {X -70.5626,Y -12.6212,Z 78,A -174.6844,B 24.896,C -2.3537,E1 24.8427,E2 -100.9772} C_DIS
LIN {X -69.8932,Y -15.9174,Z 78,A -172.0856,B 24.8969,C -2.3435,E1 24.8442,E2 -103.5669} C_DIS
LIN {X -68.8202,Y -20.0566,Z 78,A -168.2294,B 24.8969,C -2.3431,E1 24.8471,E2 -107.4446} C_DIS
LIN {X -67.5155,Y -24.0838,Z 78,A -165.0727,B 24.8983,C -2.3281,E1 24.8499,E2 -110.5832} C_DIS
LIN {X -66.1112,Y -27.7073,Z 78,A -161.6303,B 24.8984,C -2.3269,E1 24.8536,E2 -114.042} C_DIS
LIN {X -64.4509,Y -31.3782,Z 78,A -158.8586,B 24.9001,C -2.3077,E1 24.8569,E2 -116.7829} C_DIS
LIN {X -62.196,Y -35.6376,Z 78,A -154.9613,B 24.9009,C -2.2984,E1 24.8621,E2 -120.6785} C_DIS
LIN {X -60.3641,Y -38.6595,Z 78,A -152.1132,B 24.9015,C -2.2916,E1 24.8663,E2 -123.525} C_DIS
LIN {X -58.521,Y -41.3974,Z 78,A -149.2156,B 24.9015,C -2.2911,E1 24.8709,E2 -126.4356} C_DIS
LIN {X -56.0963,Y -44.6277,Z 78,A -146.3014,B 24.9028,C -2.2761,E1 24.8758,E2 -129.3279} C_DIS
LIN {X -54.1771,Y -46.9392,Z 78,A -144.007,B 24.9035,C -2.2681,E1 24.8799,E2 -131.6139} C_DIS
LIN {X -52.6697,Y -48.6243,Z 78,A -142.3153,B 24.9041,C -2.2615,E1 24.8831,E2 -133.2972} C_DIS
LIN {X -50.3477,Y -51.0243,Z 78,A -139.4767,B 24.9041,C -2.2598,E1 24.8887,E2 -136.144} C_DIS
LIN {X -48.774,Y -52.5313,Z 78,A -137.1048,B 24.9032,C -2.2713,E1 24.8936,E2 -138.5528} C_DIS
LIN {X -45.9571,Y -55.0123,Z 78,A -134.6135,B 24.9047,C -2.2534,E1 24.8988,E2 -141.0113} C_DIS
LIN {X -43.4522,Y -57.0125,Z 78,A -132.2937,B 24.9056,C -2.2431,E1 24.9039,E2 -143.315} C_DIS
LIN {X -41.1732,Y -58.6791,Z 78,A -129.6931,B 24.9052,C -2.2476,E1 24.9098,E2 -145.9353} C_DIS
LIN {X -38.006,Y -60.7776,Z 78,A -126.5556,B 24.9054,C -2.2454,E1 24.9172,E2 -149.0777} C_DIS
LIN {X -34.6164,Y -62.7712,Z 78,A -123.7077,B 24.9064,C -2.2338,E1 24.9241,E2 -151.9065} C_DIS
LIN {X -32.1972,Y -64.0458,Z 78,A -121.1625,B 24.9059,C -2.2399,E1 24.9304,E2 -154.473} C_DIS
LIN {X -27.4604,Y -66.2153,Z 78,A -117.5139,B 24.9073,C -2.2227,E1 24.9397,E2 -158.0894} C_DIS
LIN {X -22.8339,Y -67.9482,Z 78,A -112.864,B 24.9062,C -2.2367,E1 24.952,E2 -162.782} C_DIS
LIN {X -19.0389,Y -69.1088,Z 78,A -110.1004,B 24.9072,C -2.2243,E1 24.9593,E2 -165.5206} C_DIS
LIN {X -16.472,Y -69.7651,Z 78,A -107.8925,B 24.9071,C -2.2254,E1 24.9653,E2 -167.7344} C_DIS
LIN {X -11.4509,Y -70.7629,Z 78,A -104.1134,B 24.9079,C -2.216,E1 24.9757,E2 -171.495} C_DIS
LIN {X -9.3461,Y -71.0707,Z 78,A -101.6475,B 24.9063,C -2.2353,E1 24.9826,E2 -174.0086} C_DIS
LIN {X -5.4444,Y -71.4756,Z 78,A -98.2206,B 24.9056,C -2.2428,E1 24.9922,E2 -177.4549} C_DIS
LIN {X -1.7879,Y -71.6613,Z 78,A -96.3463,B 24.9079,C -2.2157,E1 24.9973,E2 -179.2652} C_DIS
LIN {X 0.4083,Y -71.6761,Z 78,A -93.3356,B 24.9051,C -2.2492,E1 25.0059,E2 -182.355} C_DIS
Enddeposition()
LIN {X 0.4083,Y -71.6761,Z 78,A -93.3356,B 24.9051,C -2.2492,E1 25.0059,E2 -182.355} C_DIS
Startdeposition()
$VEL.CP = VEL_PRINT
LIN {X -1.1606,Y -70.7419,Z 78,A -96.5417,B 24.908,C -2.2146,E1 24.9967,E2 -179.0671} C_DIS
LIN {X -4.4902,Y -70.6092,Z 78,A -99.78,B 24.9091,C -2.2009,E1 24.9876,E2 -175.7955} C_DIS
LIN {X -8.1917,Y -70.2755,Z 78,A -102.5281,B 24.9086,C -2.2077,E1 24.98,E2 -173.062} C_DIS
LIN {X -11.4245,Y -69.8233,Z 78,A -104.7482,B 24.9077,C -2.2188,E1 24.9739,E2 -170.8663} C_DIS
LIN {X -14.1074,Y -69.3307,Z 78,A -107.6091,B 24.9089,C -2.2037,E1 24.966,E2 -167.9663} C_DIS
LIN {X -17.7821,Y -68.4805,Z 78,A -110.4283,B 24.9083,C -2.211,E1 24.9584,E2 -165.1607} C_DIS
LIN {X -20.2752,Y -67.7841,Z 78,A -113.3487,B 24.9098,C -2.1927,E1 24.9504,E2 -162.1918} C_DIS
LIN {X -23.8184,Y -66.6223,Z 78,A -115.6227,B 24.9081,C -2.2129,E1 24.9445,E2 -159.9615} C_DIS
LIN {X -26.5116,Y -65.5966,Z 78,A -118.5135,B 24.909,C -2.202,E1 24.937,E2 -157.0384} C_DIS
LIN {X -29.4785,Y -64.319,Z 78,A -120.6091,B 24.9078,C -2.2171,E1 24.9317,E2 -154.9735} C_DIS
LIN {X -32.5367,Y -62.8272,Z 78,A -123.3291,B 24.9074,C -2.2213,E1 24.9249,E2 -152.2564} C_DIS
LIN {X -34.4089,Y -61.8206,Z 78,A -125.9359,B 24.909,C -2.2031,E1 24.9185,E2 -149.5986} C_DIS
LIN {X -37.8203,Y -59.7937,Z 78,A -128.3959,B 24.9071,C -2.2252,E1 24.9127,E2 -147.1836} C_DIS
LIN {X -40.3209,Y -58.1376,Z 78,A -130.4397,B 24.906,C -2.238,E1 24.9081,E2 -145.1635} C_DIS
LIN {X -42.4139,Y -56.6288,Z 78,A -132.6511,B 24.906,C -2.2387,E1 24.9031,E2 -142.9459} C_DIS
LIN {X -44.6556,Y -54.8785,Z 78,A -135.0271,B 24.9058,C -2.2412,E1 24.8979,E2 -140.5669} C_DIS
LIN {X -47.4249,Y -52.5039,Z 78,A -138.1042,B 24.9055,C -2.2441,E1 24.8914,E2 -137.4846} C_DIS
LIN {X -50.7718,Y -49.2746,Z 78,A -141.7987,B 24.9047,C -2.2535,E1 24.8841,E2 -133.797} C_DIS
LIN {X -53.2293,Y -46.6089,Z 78,A -144.796,B 24.9043,C -2.2586,E1 24.8785,E2 -130.7986} C_DIS
LIN {X -55.2392,Y -44.2105,Z 78,A -147.3517,B 24.9038,C -2.264,E1 24.8739,E2 -128.2438} C_DIS
LIN {X -56.5343,Y -42.5397,Z 78,A -149.0373,B 24.9034,C -2.2687,E1 24.8711,E2 -126.5613} C_DIS
LIN {X -58.8656,Y -39.2518,Z 78,A -152.8262,B 24.9037,C -2.2652,E1 24.8651,E2 -122.7455} C_DIS
LIN {X -60.5416,Y -36.6126,Z 78,A -155.9116,B 24.9042,C -2.2598,E1 24.8606,E2 -119.6312} C_DIS
LIN {X -62.6289,Y -32.9146,Z 78,A -158.356,B 24.9016,C -2.2906,E1 24.8574,E2 -117.2474} C_DIS
LIN {X -63.839,Y -30.5017,Z 78,A -160.311,B 24.9006,C -2.3017,E1 24.8551,E2 -115.3083} C_DIS
LIN {X -65.072,Y -27.7756,Z 78,A -163.9685,B 24.9023,C -2.2818,E1 24.8509,E2 -111.5832} C_DIS
LIN {X -66.5875,Y -23.9161,Z 78,A -166.3386,B 24.8996,C -2.3128,E1 24.8487,E2 -109.2736} C_DIS
LIN {X -67.4472,Y -21.3676,Z 78,A -168.7493,B 24.8996,C -2.3142,E1 24.8466,E2 -106.8525} C_DIS
LIN {X -68.6032,Y -17.3045,Z 78,A -171.9442,B 24.8982,C -2.3293,E1 24.8443,E2 -103.6751} C_DIS
LIN {X -69.2015,Y -14.7317,Z 78,A -174.0163,B 24.8975,C -2.3373,E1 24.843,E2 -101.6098} C_DIS
LIN {X -69.6643,Y -12.3557,Z 78,A -176.0893,B 24.8972,C -2.3409,E1 24.842,E2 -99.5333} C_DIS
LIN {X -70.0788,Y -9.7344,Z 78,A -178.1234,B 24.8964,C -2.35,E1 24.8411,E2 -97.5089} C_DIS
LIN {X -70.4268,Y -6.7738,Z 78,A 179.2036,B 24.8962,C -2.352,E1 24.8403,E2 -94.8246} C_DIS
LIN {X -70.6106,Y -4.4705,Z 78,A 177.4199,B 24.8955,C -2.3598,E1 24.84,E2 -93.0487} C_DIS
LIN {X -70.7317,Y -1.7026,Z 78,A 175.2166,B 24.8948,C -2.3677,E1 24.8398,E2 -90.8512} C_DIS
LIN {X -70.7481,Y 0.7512,Z 78,A 173.033,B 24.8946,C -2.3698,E1 24.8398,E2 -88.6595} C_DIS
LIN {X -70.6154,Y 4.3997,Z 78,A 170.2355,B 24.8935,C -2.3826,E1 24.8402,E2 -85.8757} C_DIS
LIN {X -70.3618,Y 7.414,Z 78,A 167.4581,B 24.8934,C -2.3834,E1 24.8409,E2 -83.0835} C_DIS
LIN {X -69.8297,Y 11.3864,Z 78,A 164.8059,B 24.8913,C -2.4064,E1 24.842,E2 -80.4703} C_DIS
LIN {X -69.4582,Y 13.4651,Z 78,A 162.6406,B 24.8917,C -2.402,E1 24.8431,E2 -78.2818} C_DIS
LIN {X -68.7464,Y 16.7237,Z 78,A 159.9806,B 24.8909,C -2.4114,E1 24.8448,E2 -75.6285} C_DIS
LIN {X -67.7309,Y 20.4548,Z 78,A 156.5158,B 24.8906,C -2.414,E1 24.8474,E2 -72.1499} C_DIS
LIN {X -66.6885,Y 23.6313,Z 78,A 154.1318,B 24.8893,C -2.4292,E1 24.8496,E2 -69.7886} C_DIS
LIN {X -65.6268,Y 26.4374,Z 78,A 151.6539,B 24.8887,C -2.4355,E1 24.8521,E2 -67.3119} C_DIS
LIN {X -64.6057,Y 28.8428,Z 78,A 149.1567,B 24.8888,C -2.4336,E1 24.8549,E2 -64.7965} C_DIS
LIN {X -63.1299,Y 31.9444,Z 78,A 146.992,B 24.8869,C -2.4551,E1 24.8575,E2 -62.6714} C_DIS
LIN {X -61.8519,Y 34.3529,Z 78,A 144.298,B 24.8873,C -2.4509,E1 24.8612,E2 -59.9532} C_DIS
LIN {X -60.3704,Y 36.8943,Z 78,A 141.7167,B 24.887,C -2.4534,E1 24.8649,E2 -57.3644} C_DIS
LIN {X -57.7512,Y 40.8732,Z 78,A 138.3386,B 24.8851,C -2.4743,E1 24.8701,E2 -54.0195} C_DIS
LIN {X -55.8727,Y 43.4058,Z 78,A 135.3118,B 24.8854,C -2.4707,E1 24.8753,E2 -50.9698} C_DIS
LIN {X -52.2066,Y 47.7518,Z 78,A 131.0152,B 24.8837,C -2.4891,E1 24.8831,E2 -46.6976} C_DIS
LIN {X -50.0933,Y 49.9653,Z 78,A 128.7274,B 24.8828,C -2.4993,E1 24.8875,E2 -44.4243} C_DIS
LIN {X -47.0444,Y 52.8452,Z 78,A 124.6178,B 24.8835,C -2.4913,E1 24.8961,E2 -40.279} C_DIS
LIN {X -42.8613,Y 56.2923,Z 78,A 120.6489,B 24.8817,C -2.51,E1 24.9047,E2 -36.3398} C_DIS
LIN {X -40.0786,Y 58.3053,Z 78,A 117.8586,B 24.8812,C -2.5153,E1 24.911,E2 -33.5527} C_DIS
LIN {X -37.8167,Y 59.798,Z 78,A 115.1754,B 24.8819,C -2.5084,E1 24.9174,E2 -30.8445} C_DIS
LIN {X -34.6055,Y 61.7108,Z 78,A 112.6963,B 24.8802,C -2.5261,E1 24.9233,E2 -28.4001} C_DIS
LIN {X -31.9017,Y 63.1517,Z 78,A 110.1261,B 24.88,C -2.5281,E1 24.9297,E2 -25.8278} C_DIS
LIN {X -29.205,Y 64.4425,Z 78,A 107.8617,B 24.8793,C -2.5354,E1 24.9354,E2 -23.575} C_DIS
LIN {X -26.4928,Y 65.6043,Z 78,A 104.8802,B 24.8803,C -2.5251,E1 24.9432,E2 -20.5623} C_DIS
LIN {X -22.5709,Y 67.0545,Z 78,A 102.1233,B 24.8785,C -2.5439,E1 24.9503,E2 -17.8447} C_DIS
LIN {X -17.603,Y 68.5265,Z 78,A 97.9114,B 24.8781,C -2.548,E1 24.9616,E2 -13.6356} C_DIS
LIN {X -14.9565,Y 69.1525,Z 78,A 95.5605,B 24.8783,C -2.5464,E1 24.968,E2 -11.278} C_DIS
LIN {X -12.0251,Y 69.7228,Z 78,A 93.4383,B 24.8774,C -2.5553,E1 24.9738,E2 -9.1747} C_DIS
LIN {X -9.0156,Y 70.1746,Z 78,A 90.8965,B 24.8774,C -2.5551,E1 24.9808,E2 -6.6302} C_DIS
LIN {X -5.4728,Y 70.5395,Z 78,A 87.865,B 24.8776,C -2.5529,E1 24.9893,E2 -3.5921} C_DIS
LIN {X -2.6283,Y 70.7037,Z 78,A 85.4306,B 24.8779,C -2.5506,E1 24.9961,E2 -1.1516} C_DIS
LIN {X -0.6042,Y 70.7489,Z 78,A 83.6463,B 24.8782,C -2.5475,E1 25.0011,E2 0.6401} C_DIS
LIN {X 3.7978,Y 70.6494,Z 78,A 80.2205,B 24.8778,C -2.5512,E1 25.0106,E2 4.0563} C_DIS
LIN {X 6.8563,Y 70.4192,Z 78,A 77.7681,B 24.8778,C -2.5518,E1 25.0174,E2 6.506} C_DIS
LIN {X 10.7839,Y 69.9246,Z 78,A 74.4082,B 24.8782,C -2.5472,E1 25.0268,E2 9.8738} C_DIS
LIN {X 14.0509,Y 69.3423,Z 78,A 71.8923,B 24.8779,C -2.5504,E1 25.0336,E2 12.3792} C_DIS
LIN {X 17.0736,Y 68.661,Z 78,A 69.1817,B 24.8785,C -2.544,E1 25.041,E2 15.1012} C_DIS
LIN {X 20.8216,Y 67.6179,Z 78,A 66.1451,B 24.8785,C -2.5447,E1 25.0491,E2 18.131} C_DIS
LIN {X 23.5359,Y 66.722,Z 78,A 63.075,B 24.8805,C -2.5236,E1 25.0574,E2 21.2449} C_DIS
LIN {X 27.071,Y 65.3689,Z 78,A 60.7822,B 24.8789,C -2.5401,E1 25.0632,E2 23.4933} C_DIS
LIN {X 30.1538,Y 64.0047,Z 78,A 58.1209,B 24.879,C -2.5388,E1 25.0699,E2 26.1511} C_DIS
LIN {X 33.8025,Y 62.1538,Z 78,A 54.1378,B 24.8811,C -2.5172,E1 25.0798,E2 30.1741} C_DIS
LIN {X 36.72,Y 60.4764,Z 78,A 52.1303,B 24.8797,C -2.5318,E1 25.0846,E2 32.1407} C_DIS
LIN {X 40.148,Y 58.2578,Z 78,A 48.8721,B 24.88,C -2.5279,E1 25.0921,E2 35.3976} C_DIS
LIN {X 42.4906,Y 56.5712,Z 78,A 46.476,B 24.8806,C -2.5223,E1 25.0975,E2 37.7983} C_DIS
LIN {X 44.9575,Y 54.6323,Z 78,A 43.9521,B 24.881,C -2.5181,E1 25.103,E2 40.3227} C_DIS
LIN {X 47.1777,Y 52.7258,Z 78,A 41,B 24.8829,C -2.4981,E1 25.1093,E2 43.3104} C_DIS
LIN {X 49.8524,Y 50.2048,Z 78,A 38.2013,B 24.883,C -2.4966,E1 25.1148,E2 46.1009} C_DIS
LIN {X 52.6811,Y 47.2276,Z 78,A 35.348,B 24.8825,C -2.5019,E1 25.1202,E2 48.929} C_DIS
LIN {X 54.6878,Y 44.8907,Z 78,A 32.8756,B 24.883,C -2.4968,E1 25.1246,E2 51.4023} C_DIS
LIN {X 56.4291,Y 42.6797,Z 78,A 30.6893,B 24.8833,C -2.4939,E1 25.1284,E2 53.5851} C_DIS
LIN {X 58.9342,Y 39.148,Z 78,A 27.2475,B 24.8839,C -2.4869,E1 25.1339,E2 57.0265} C_DIS
LIN {X 61.5676,Y 34.8619,Z 78,A 23.0343,B 24.8853,C -2.4724,E1 25.14,E2 61.2524} C_DIS
LIN {X 63.0002,Y 32.1982,Z 78,A 20.6544,B 24.8857,C -2.4677,E1 25.143,E2 63.6309} C_DIS
LIN {X 63.9884,Y 30.1887,Z 78,A 18.7867,B 24.8863,C -2.4612,E1 25.1453,E2 65.504} C_DIS
LIN {X 66.1142,Y 25.1929,Z 78,A 14.6407,B 24.8868,C -2.4556,E1 25.1497,E2 69.6404} C_DIS
LIN {X 67.241,Y 22.0102,Z 78,A 11.7829,B 24.8879,C -2.4441,E1 25.1523,E2 72.5092} C_DIS
LIN {X 68.075,Y 19.2755,Z 78,A 9.4515,B 24.8886,C -2.4368,E1 25.1542,E2 74.8447} C_DIS
LIN {X 68.6971,Y 16.9257,Z 78,A 7.2578,B 24.8897,C -2.4245,E1 25.1557,E2 77.0546} C_DIS
LIN {X 69.6779,Y 12.2799,Z 78,A 3.6332,B 24.8902,C -2.4189,E1 25.1577,E2 80.6714} C_DIS
LIN {X 70.1486,Y 9.2165,Z 78,A 1.4751,B 24.89,C -2.4209,E1 25.1585,E2 82.812} C_DIS
LIN {X 70.5002,Y 5.9652,Z 78,A -1.8039,B 24.8924,C -2.3949,E1 25.1594,E2 86.1329} C_DIS
LIN {X 70.7247,Y 1.9528,Z 78,A -4.6264,B 24.8922,C -2.3967,E1 25.1598,E2 88.9344} C_DIS
LIN {X 70.7487,Y -0.6505,Z 78,A -6.5539,B 24.8923,C -2.3951,E1 25.1598,E2 90.8543} C_DIS
LIN {X 70.6027,Y -4.587,Z 78,A -9.9057,B 24.8937,C -2.3804,E1 25.1594,E2 94.2209} C_DIS
LIN {X 70.1104,Y -9.5111,Z 78,A -14.0328,B 24.8951,C -2.3643,E1 25.1581,E2 98.3616} C_DIS
LIN {X 69.4928,Y -13.2855,Z 78,A -17.4922,B 24.8969,C -2.3444,E1 25.1564,E2 101.8478} C_DIS
LIN {X 68.5894,Y -17.3584,Z 78,A -20.2851,B 24.8964,C -2.3502,E1 25.1546,E2 104.6109} C_DIS
LIN {X 67.7961,Y -20.2348,Z 78,A -22.9393,B 24.8976,C -2.336,E1 25.1525,E2 107.2833} C_DIS
LIN {X 66.831,Y -23.2252,Z 78,A -25.148,B 24.8975,C -2.3376,E1 25.1506,E2 109.4759} C_DIS
LIN {X 65.7743,Y -26.0678,Z 78,A -28.0501,B 24.8992,C -2.3176,E1 25.1476,E2 112.409} C_DIS
LIN {X 63.6333,Y -30.9298,Z 78,A -32.5128,B 24.9007,C -2.3004,E1 25.1424,E2 116.8882} C_DIS
LIN {X 61.5741,Y -34.8502,Z 78,A -35.9773,B 24.9013,C -2.2934,E1 25.1377,E2 120.3513} C_DIS
LIN {X 59.7034,Y -37.9651,Z 78,A -39.6265,B 24.9037,C -2.2657,E1 25.1322,E2 124.0473} C_DIS
LIN {X 57.1986,Y -41.6425,Z 78,A -41.6904,B 24.9009,C -2.2983,E1 25.129,E2 126.0243} C_DIS
LIN {X 56.1943,Y -42.9878,Z 78,A -43.8316,B 24.9031,C -2.2731,E1 25.1253,E2 128.2149} C_DIS
LIN {X 53.5013,Y -46.2975,Z 78,A -47.6049,B 24.9046,C -2.2555,E1 25.1185,E2 132.0125} C_DIS
LIN {X 51.2157,Y -48.8127,Z 78,A -49.7713,B 24.9038,C -2.2647,E1 25.1144,E2 134.1477} C_DIS
LIN {X 48.4274,Y -51.5804,Z 78,A -52.8194,B 24.9041,C -2.2608,E1 25.1082,E2 137.1924} C_DIS
LIN {X 46.1561,Y -53.6236,Z 78,A -54.9359,B 24.9038,C -2.2649,E1 25.1039,E2 139.2907} C_DIS
LIN {X 42.7254,Y -56.3941,Z 78,A -58.6558,B 24.9048,C -2.2531,E1 25.0957,E2 143.0246} C_DIS
LIN {X 41.1953,Y -57.5214,Z 78,A -60.8456,B 24.9065,C -2.2325,E1 25.0907,E2 145.2555} C_DIS
LIN {X 37.8501,Y -59.7771,Z 78,A -63.4669,B 24.9056,C -2.2435,E1 25.0846,E2 147.8422} C_DIS
LIN {X 34.549,Y -61.7423,Z 78,A -66.3651,B 24.9056,C -2.2435,E1 25.0776,E2 150.7312} C_DIS
LIN {X 32.0042,Y -63.0993,Z 78,A -69.1923,B 24.907,C -2.2266,E1 25.0706,E2 153.5909} C_DIS
LIN {X 28.1443,Y -64.9128,Z 78,A -72.2161,B 24.9065,C -2.2327,E1 25.0629,E2 156.5926} C_DIS
LIN {X 23.943,Y -66.5777,Z 78,A -76.2007,B 24.9076,C -2.2191,E1 25.0525,E2 160.6005} C_DIS
LIN {X 20.5613,Y -67.699,Z 78,A -79.0594,B 24.9078,C -2.2164,E1 25.0449,E2 163.4604} C_DIS
LIN {X 17.1157,Y -68.6508,Z 78,A -82.2601,B 24.9088,C -2.2056,E1 25.0362,E2 166.6819} C_DIS
LIN {X 12.9496,Y -69.5575,Z 78,A -85.3532,B 24.9082,C -2.2118,E1 25.0278,E2 169.7564} C_DIS
LIN {X 10.0708,Y -70.031,Z 78,A -87.3052,B 24.9075,C -2.2207,E1 25.0225,E2 171.6854} C_DIS
LIN {X 5.8385,Y -70.5103,Z 78,A -90.9567,B 24.9081,C -2.2136,E1 25.0123,E2 175.3514} C_DIS
LIN {X 1.7707,Y -70.7302,Z 78,A -94.4742,B 24.9086,C -2.2068,E1 25.0024,E2 178.8839} C_DIS
LIN {X 1.7707,Y -70.7302,Z 78,A -94.4742,B 24.9086,C -2.2068,E1 25.0024,E2 178.8839} C_DIS
Enddeposition()
LIN {X 0.3843,Y -69.8184,Z 78,A -94.5954,B 24.9052,C -2.248,E1 25.0024,E2 178.9073} C_DIS
Startdeposition()
$VEL.CP = VEL_PRINT
LIN {X 3.3748,Y -69.7396,Z 78,A -91.878,B 24.9046,C -2.2555,E1 25.01,E2 176.1728} C_DIS
LIN {X 6.7049,Y -69.4981,Z 78,A -89.1101,B 24.9044,C -2.2576,E1 25.0177,E2 173.4015} C_DIS
LIN {X 9.6724,Y -69.1471,Z 78,A -86.8135,B 24.9046,C -2.2551,E1 25.024,E2 171.1125} C_DIS
LIN {X 12.5857,Y -68.6769,Z 78,A -84.2807,B 24.9042,C -2.2599,E1 25.031,E2 168.5712} C_DIS
LIN {X 15.5466,Y -68.0675,Z 78,A -81.5997,B 24.9036,C -2.2673,E1 25.0384,E2 165.876} C_DIS
LIN {X 18.6337,Y -67.289,Z 78,A -79.252,B 24.9039,C -2.2631,E1 25.0447,E2 163.5422} C_DIS
LIN {X 21.3777,Y -66.467,Z 78,A -77.0089,B 24.9039,C -2.2631,E1 25.0506,E2 161.3033} C_DIS
LIN {X 23.9927,Y -65.5684,Z 78,A -74.4278,B 24.903,C -2.2742,E1 25.0575,E2 158.7009} C_DIS
LIN {X 27.0204,Y -64.3798,Z 78,A -72.013,B 24.9032,C -2.2712,E1 25.0637,E2 156.2988} C_DIS
LIN {X 29.6073,Y -63.232,Z 78,A -69.6631,B 24.9029,C -2.2755,E1 25.0697,E2 153.9446} C_DIS
LIN {X 33.9476,Y -61.0117,Z 78,A -65.8375,B 24.9027,C -2.2775,E1 25.0791,E2 150.125} C_DIS
LIN {X 36.1922,Y -59.7075,Z 78,A -63.6812,B 24.9023,C -2.282,E1 25.0843,E2 147.9646} C_DIS
LIN {X 38.5253,Y -58.2295,Z 78,A -60.9021,B 24.9007,C -2.3003,E1 25.0909,E2 145.1514} C_DIS
LIN {X 41.9033,Y -55.8478,Z 78,A -56.966,B 24.8988,C -2.3223,E1 25.0998,E2 141.1773} C_DIS
LIN {X 45.0713,Y -53.3246,Z 78,A -55.0008,B 24.9014,C -2.2922,E1 25.1039,E2 139.2907} C_DIS
LIN {X 47.5445,Y -51.1325,Z 78,A -51.8886,B 24.8999,C -2.3094,E1 25.1104,E2 136.1504} C_DIS
LIN {X 49.6372,Y -49.102,Z 78,A -48.336,B 24.8966,C -2.3475,E1 25.1175,E2 132.5229} C_DIS
LIN {X 52.825,Y -45.6563,Z 78,A -45.9157,B 24.8993,C -2.3172,E1 25.1218,E2 130.185} C_DIS
LIN {X 54.5298,Y -43.6063,Z 78,A -43.2145,B 24.8975,C -2.3372,E1 25.1266,E2 127.449} C_DIS
LIN {X 56.8498,Y -40.5334,Z 78,A -39.542,B 24.8955,C -2.3601,E1 25.1327,E2 123.7401} C_DIS
LIN {X 58.9651,Y -37.3914,Z 78,A -37.3347,B 24.897,C -2.3435,E1 25.136,E2 121.5833} C_DIS
LIN {X 60.3523,Y -35.1083,Z 78,A -35.2183,B 24.8966,C -2.3476,E1 25.139,E2 119.468} C_DIS
LIN {X 61.5421,Y -32.978,Z 78,A -32.5053,B 24.8943,C -2.3734,E1 25.1426,E2 116.7082} C_DIS
LIN {X 63.7708,Y -28.4293,Z 78,A -28.9559,B 24.8947,C -2.3686,E1 25.1468,E2 113.1894} C_DIS
LIN {X 65.006,Y -25.4771,Z 78,A -26.4315,B 24.8943,C -2.3737,E1 25.1494,E2 110.667} C_DIS
LIN {X 66.5642,Y -21.0737,Z 78,A -22.8076,B 24.8937,C -2.3795,E1 25.1527,E2 107.0496} C_DIS
LIN {X 67.2617,Y -18.73,Z 78,A -20.6072,B 24.8927,C -2.3912,E1 25.1544,E2 104.8342} C_DIS
LIN {X 67.9804,Y -15.9236,Z 78,A -18.3035,B 24.8922,C -2.3966,E1 25.1559,E2 102.5311} C_DIS
LIN {X 68.508,Y -13.4756,Z 78,A -16.2943,B 24.8917,C -2.4018,E1 25.1571,E2 100.5213} C_DIS
LIN {X 68.9349,Y -11.091,Z 78,A -14.2595,B 24.8911,C -2.4094,E1 25.158,E2 98.4805} C_DIS
LIN {X 69.3398,Y -8.1759,Z 78,A -11.7107,B 24.89,C -2.4209,E1 25.1589,E2 95.9197} C_DIS
LIN {X 69.6285,Y -5.184,Z 78,A -9.4727,B 24.8899,C -2.4222,E1 25.1594,E2 93.6917} C_DIS
LIN {X 69.7778,Y -2.451,Z 78,A -7.4962,B 24.8899,C -2.4218,E1 25.1597,E2 91.7279} C_DIS
LIN {X 69.8184,Y -0.518,Z 78,A -5.7069,B 24.8889,C -2.4326,E1 25.1597,E2 89.9239} C_DIS
LIN {X 69.7905,Y 2.0383,Z 78,A -3.6143,B 24.8884,C -2.4391,E1 25.1597,E2 87.8284} C_DIS
LIN {X 69.6343,Y 5.1072,Z 78,A -1.033,B 24.8875,C -2.4487,E1 25.1592,E2 85.2397} C_DIS
LIN {X 69.4011,Y 7.6476,Z 78,A 1.2077,B 24.8865,C -2.4594,E1 25.1586,E2 82.987} C_DIS
LIN {X 69.0138,Y 10.5808,Z 78,A 3.3889,B 24.8865,C -2.46,E1 25.1577,E2 80.8172} C_DIS
LIN {X 68.4737,Y 13.6506,Z 78,A 6.0203,B 24.8855,C -2.4699,E1 25.1564,E2 78.1777} C_DIS
LIN {X 67.8254,Y 16.5703,Z 78,A 8.4072,B 24.885,C -2.4755,E1 25.1549,E2 75.7913} C_DIS
LIN {X 67.1263,Y 19.2081,Z 78,A 10.6321,B 24.8844,C -2.4819,E1 25.1532,E2 73.5643} C_DIS
LIN {X 66.3372,Y 21.779,Z 78,A 12.8073,B 24.8839,C -2.4875,E1 25.1514,E2 71.3881} C_DIS
LIN {X 65.4135,Y 24.4141,Z 78,A 15.7662,B 24.8815,C -2.5128,E1 25.1485,E2 68.3859} C_DIS
LIN {X 63.8546,Y 28.2414,Z 78,A 18.3632,B 24.8827,C -2.5003,E1 25.1457,E2 65.8327} C_DIS
LIN {X 62.7092,Y 30.7006,Z 78,A 20.654,B 24.8819,C -2.5083,E1 25.1429,E2 63.5355} C_DIS
LIN {X 61.6592,Y 32.7576,Z 78,A 22.4913,B 24.8816,C -2.5118,E1 25.1405,E2 61.6995} C_DIS
LIN {X 60.5515,Y 34.7617,Z 78,A 24.5463,B 24.8806,C -2.5217,E1 25.1377,E2 59.6318} C_DIS
LIN {X 58.5459,Y 38.0445,Z 78,A 27.3624,B 24.8808,C -2.5205,E1 25.1336,E2 56.8328} C_DIS
LIN {X 56.3866,Y 41.1755,Z 78,A 30.6397,B 24.8796,C -2.5325,E1 25.1283,E2 53.5432} C_DIS
LIN {X 54.5424,Y 43.5904,Z 78,A 33.31,B 24.8786,C -2.5432,E1 25.1237,E2 50.8601} C_DIS
LIN {X 52.341,Y 46.2106,Z 78,A 36.0963,B 24.878,C -2.549,E1 25.1186,E2 48.0727} C_DIS
LIN {X 50.0725,Y 48.6588,Z 78,A 38.807,B 24.8775,C -2.5541,E1 25.1134,E2 45.3616} C_DIS
LIN {X 47.4303,Y 51.2378,Z 78,A 41.8062,B 24.877,C -2.5595,E1 25.1073,E2 42.3621} C_DIS
LIN {X 44.9303,Y 53.4442,Z 78,A 44.4769,B 24.8767,C -2.563,E1 25.1017,E2 39.6936} C_DIS
LIN {X 42.8028,Y 55.1619,Z 78,A 46.8091,B 24.8761,C -2.5694,E1 25.0966,E2 37.3548} C_DIS
LIN {X 40.3363,Y 56.9905,Z 78,A 49.1815,B 24.8761,C -2.5698,E1 25.0912,E2 34.9899} C_DIS
LIN {X 37.9692,Y 58.5943,Z 78,A 51.6603,B 24.8753,C -2.577,E1 25.0854,E2 32.5023} C_DIS
LIN {X 35.1859,Y 60.3051,Z 78,A 55.1636,B 24.8728,C -2.6026,E1 25.0769,E2 28.9489} C_DIS
LIN {X 31.7551,Y 62.181,Z 78,A 57.2859,B 24.8752,C -2.5782,E1 25.0718,E2 26.8904} C_DIS
LIN {X 29.0448,Y 63.4934,Z 78,A 59.994,B 24.8743,C -2.5872,E1 25.0649,E2 24.1679} C_DIS
LIN {X 26.4414,Y 64.6199,Z 78,A 62.0701,B 24.8747,C -2.5832,E1 25.0596,E2 22.1062} C_DIS
LIN {X 23.9912,Y 65.5689,Z 78,A 64.3336,B 24.8743,C -2.588,E1 25.0536,E2 19.8363} C_DIS
LIN {X 21.7706,Y 66.3398,Z 78,A 66.7077,B 24.873,C -2.6009,E1 25.0473,E2 17.436} C_DIS
LIN {X 16.8835,Y 67.749,Z 78,A 70.4425,B 24.8738,C -2.5924,E1 25.0373,E2 13.7274} C_DIS
LIN {X 14.2805,Y 68.3446,Z 78,A 72.6081,B 24.8738,C -2.5928,E1 25.0314,E2 11.5637} C_DIS
LIN {X 11.6341,Y 68.8442,Z 78,A 74.9129,B 24.8735,C -2.596,E1 25.025,E2 9.2537} C_DIS
LIN {X 9.0095,Y 69.2365,Z 78,A 76.9279,B 24.8738,C -2.5925,E1 25.0195,E2 7.2489} C_DIS
LIN {X 6.3854,Y 69.5276,Z 78,A 79.0783,B 24.8738,C -2.5924,E1 25.0135,E2 5.1002} C_DIS
LIN {X 3.7897,Y 69.7173,Z 78,A 81.3177,B 24.8736,C -2.5949,E1 25.0073,E2 2.8556} C_DIS
LIN {X 0.6698,Y 69.8174,Z 78,A 83.9599,B 24.8734,C -2.5966,E1 24.9999,E2 0.2099} C_DIS
LIN {X -2.3359,Y 69.7814,Z 78,A 86.3323,B 24.8737,C -2.5936,E1 24.9933,E2 -2.1557} C_DIS
LIN {X -5.002,Y 69.6414,Z 78,A 88.6034,B 24.8736,C -2.5947,E1 24.9869,E2 -4.4301} C_DIS
LIN {X -8.2866,Y 69.3269,Z 78,A 91.1756,B 24.8741,C -2.59,E1 24.9798,E2 -6.9927} C_DIS
LIN {X -10.861,Y 68.9705,Z 78,A 93.1095,B 24.8747,C -2.5839,E1 24.9745,E2 -8.9136} C_DIS
LIN {X -12.8132,Y 68.6355,Z 78,A 95.0346,B 24.8741,C -2.5898,E1 24.9692,E2 -10.8547} C_DIS
LIN {X -15.4094,Y 68.0992,Z 78,A 97.1854,B 24.8743,C -2.5873,E1 24.9633,E2 -13.0023} C_DIS
LIN {X -17.9584,Y 67.4716,Z 78,A 99.3128,B 24.8746,C -2.5846,E1 24.9576,E2 -15.1263} C_DIS
LIN {X -21.1114,Y 66.5532,Z 78,A 101.822,B 24.8753,C -2.5773,E1 24.9509,E2 -17.6223} C_DIS
LIN {X -23.1316,Y 65.877,Z 78,A 103.9259,B 24.8747,C -2.5835,E1 24.9453,E2 -19.745} C_DIS
LIN {X -26.2423,Y 64.7009,Z 78,A 106.4592,B 24.8755,C -2.5753,E1 24.9387,E2 -22.2642} C_DIS
LIN {X -28.5624,Y 63.7108,Z 78,A 108.5538,B 24.8757,C -2.5728,E1 24.9334,E2 -24.3579} C_DIS
LIN {X -30.8719,Y 62.6243,Z 78,A 110.656,B 24.876,C -2.5698,E1 24.9281,E2 -26.4583} C_DIS
LIN {X -33.0876,Y 61.4827,Z 78,A 112.6989,B 24.8764,C -2.5663,E1 24.9231,E2 -28.4986} C_DIS
LIN {X -35.3544,Y 60.2077,Z 78,A 115.6135,B 24.875,C -2.5805,E1 24.9159,E2 -31.4557} C_DIS
LIN {X -38.0962,Y 58.5124,Z 78,A 118.1826,B 24.8756,C -2.5737,E1 24.9099,E2 -34.017} C_DIS
LIN {X -42.1435,Y 55.6673,Z 78,A 121.7671,B 24.8775,C -2.5547,E1 24.9019,E2 -37.5688} C_DIS
LIN {X -45.0757,Y 53.3208,Z 78,A 124.8345,B 24.8782,C -2.5477,E1 24.8953,E2 -40.631} C_DIS
LIN {X -47.6806,Y 51.0045,Z 78,A 127.4163,B 24.8794,C -2.535,E1 24.89,E2 -43.1929} C_DIS
LIN {X -49.3839,Y 49.3582,Z 78,A 129.644,B 24.8792,C -2.5367,E1 24.8856,E2 -45.434} C_DIS
LIN {X -51.4696,Y 47.1778,Z 78,A 132.0869,B 24.8799,C -2.5299,E1 24.8809,E2 -47.8714} C_DIS
LIN {X -53.6766,Y 44.6506,Z 78,A 134.7524,B 24.8807,C -2.521,E1 24.8761,E2 -50.5278} C_DIS
LIN {X -54.8056,Y 43.2575,Z 78,A 137.2778,B 24.8788,C -2.5405,E1 24.8717,E2 -53.1116} C_DIS
LIN {X -57.1281,Y 40.1417,Z 78,A 139.5734,B 24.8815,C -2.5121,E1 24.868,E2 -55.3507} C_DIS
LIN {X -58.8194,Y 37.6185,Z 78,A 142.056,B 24.8822,C -2.505,E1 24.8642,E2 -57.8288} C_DIS
LIN {X -60.3805,Y 35.0593,Z 78,A 144.5098,B 24.8829,C -2.4979,E1 24.8607,E2 -60.2784} C_DIS
LIN {X -61.7353,Y 32.6131,Z 78,A 147.4458,B 24.8822,C -2.5053,E1 24.8568,E2 -63.2476} C_DIS
LIN {X -63.6295,Y 28.7427,Z 78,A 150.0484,B 24.8851,C -2.4746,E1 24.8538,E2 -65.791} C_DIS
LIN {X -64.4355,Y 26.8884,Z 78,A 152.0571,B 24.8848,C -2.4771,E1 24.8516,E2 -67.8168} C_DIS
LIN {X -65.4373,Y 24.3512,Z 78,A 154.4862,B 24.8851,C -2.4745,E1 24.8491,E2 -70.2532} C_DIS
LIN {X -66.7366,Y 20.521,Z 78,A 157.4659,B 24.8867,C -2.457,E1 24.8466,E2 -73.2081} C_DIS
LIN {X -67.7129,Y 17.0281,Z 78,A 161.109,B 24.8862,C -2.4621,E1 24.8439,E2 -76.8847} C_DIS
LIN {X -68.4692,Y 13.6734,Z 78,A 163.6367,B 24.8876,C -2.4468,E1 24.8425,E2 -79.3909} C_DIS
LIN {X -69.0275,Y 10.4925,Z 78,A 166.181,B 24.8886,C -2.4362,E1 24.8414,E2 -81.9248} C_DIS
LIN {X -69.4054,Y 7.607,Z 78,A 168.4108,B 24.8896,C -2.4252,E1 24.8406,E2 -84.1417} C_DIS
LIN {X -69.6226,Y 5.2582,Z 78,A 170.5809,B 24.8897,C -2.4241,E1 24.8401,E2 -86.3222} C_DIS
LIN {X -69.7838,Y 2.2559,Z 78,A 172.9892,B 24.8905,C -2.415,E1 24.8398,E2 -88.7233} C_DIS
LIN {X -69.8179,Y -0.601,Z 78,A 175.4169,B 24.8911,C -2.4093,E1 24.8398,E2 -91.1522} C_DIS
LIN {X -69.7325,Y -3.5138,Z 78,A 177.7946,B 24.8918,C -2.4015,E1 24.8401,E2 -93.5254} C_DIS
LIN {X -69.5335,Y -6.321,Z 78,A -179.8993,B 24.8924,C -2.3942,E1 24.8406,E2 -95.8278} C_DIS
LIN {X -69.2088,Y -9.2231,Z 78,A -177.4581,B 24.893,C -2.3877,E1 24.8414,E2 -98.2681} C_DIS
LIN {X -68.766,Y -12.0901,Z 78,A -175.1343,B 24.8938,C -2.3791,E1 24.8425,E2 -100.5852} C_DIS
LIN {X -68.2291,Y -14.8207,Z 78,A -172.8151,B 24.8943,C -2.3729,E1 24.8438,E2 -102.9032} C_DIS
LIN {X -67.6945,Y -17.0997,Z 78,A -170.5872,B 24.8943,C -2.3737,E1 24.8453,E2 -105.1462} C_DIS
LIN {X -66.4011,Y -21.5815,Z 78,A -166.9409,B 24.8956,C -2.3584,E1 24.8482,E2 -108.7768} C_DIS
LIN {X -65.3712,Y -24.5256,Z 78,A -164.4282,B 24.8964,C -2.3499,E1 24.8506,E2 -111.2835} C_DIS
LIN {X -64.0279,Y -27.8441,Z 78,A -161.4614,B 24.8971,C -2.3422,E1 24.8538,E2 -114.2484} C_DIS
LIN {X -62.757,Y -30.6036,Z 78,A -158.9358,B 24.8976,C -2.336,E1 24.8568,E2 -116.7729} C_DIS
LIN {X -61.4962,Y -33.0627,Z 78,A -156.3199,B 24.8975,C -2.3376,E1 24.8603,E2 -119.4066} C_DIS
LIN {X -59.5431,Y -36.4627,Z 78,A -153.4777,B 24.8989,C -2.3208,E1 24.8643,E2 -122.2234} C_DIS
LIN {X -57.9911,Y -38.8842,Z 78,A -150.523,B 24.8983,C -2.3282,E1 24.8689,E2 -125.2105} C_DIS
LIN {X -55.933,Y -41.7898,Z 78,A -148.1489,B 24.9,C -2.3087,E1 24.8728,E2 -127.5497} C_DIS
LIN {X -54.152,Y -44.0731,Z 78,A -145.7243,B 24.9004,C -2.3043,E1 24.877,E2 -129.9749} C_DIS
LIN {X -52.2811,Y -46.2785,Z 78,A -143.2118,B 24.9006,C -2.3021,E1 24.8816,E2 -132.4935} C_DIS
LIN {X -50.6431,Y -48.0649,Z 78,A -141.2751,B 24.901,C -2.2966,E1 24.8853,E2 -134.4256} C_DIS
LIN {X -48.0713,Y -50.6371,Z 78,A -137.8312,B 24.9007,C -2.301,E1 24.8922,E2 -137.8945} C_DIS
LIN {X -44.8008,Y -53.5518,Z 78,A -134.7509,B 24.9023,C -2.2823,E1 24.8987,E2 -140.9421} C_DIS
LIN {X -42.2907,Y -55.5565,Z 78,A -132.1496,B 24.9027,C -2.2768,E1 24.9044,E2 -143.5399} C_DIS
LIN {X -39.2424,Y -57.7487,Z 78,A -128.3681,B 24.9018,C -2.2882,E1 24.9131,E2 -147.3614} C_DIS
LIN {X -34.2014,Y -60.87,Z 78,A -124.1814,B 24.9037,C -2.2651,E1 24.9231,E2 -151.5059} C_DIS
LIN {X -31.935,Y -62.089,Z 78,A -122.0693,B 24.904,C -2.2624,E1 24.9283,E2 -153.6175} C_DIS
LIN {X -29.203,Y -63.4202,Z 78,A -119.5738,B 24.9042,C -2.2596,E1 24.9346,E2 -156.1126} C_DIS
LIN {X -26.4273,Y -64.6256,Z 78,A -117.1925,B 24.9046,C -2.2546,E1 24.9407,E2 -158.4875} C_DIS
LIN {X -24.834,Y -65.2544,Z 78,A -115.1824,B 24.9035,C -2.2679,E1 24.946,E2 -160.5334} C_DIS
LIN {X -20.1359,Y -66.8542,Z 78,A -111.5316,B 24.9046,C -2.2545,E1 24.9557,E2 -164.159} C_DIS
LIN {X -17.5119,Y -67.5885,Z 78,A -109.3406,B 24.9049,C -2.252,E1 24.9616,E2 -166.3476} C_DIS
LIN {X -14.9451,Y -68.202,Z 78,A -107.043,B 24.9047,C -2.2542,E1 24.9678,E2 -168.6534} C_DIS
LIN {X -11.7766,Y -68.8203,Z 78,A -104.4699,B 24.9049,C -2.2514,E1 24.9749,E2 -171.2224} C_DIS
LIN {X -9.1419,Y -69.2193,Z 78,A -102.3475,B 24.9051,C -2.2494,E1 24.9808,E2 -173.3417} C_DIS
LIN {X -6.6631,Y -69.5019,Z 78,A -100.2388,B 24.905,C -2.2507,E1 24.9866,E2 -175.4547} C_DIS
LIN {X -3.5233,Y -69.7314,Z 78,A -97.7101,B 24.905,C -2.2494,E1 24.9937,E2 -177.9811} C_DIS
LIN {X -1.0037,Y -69.8135,Z 78,A -95.613,B 24.905,C -2.2504,E1 24.9995,E2 -180.0809} C_DIS
LIN {X -1.0037,Y -69.8135,Z 78,A -95.613,B 24.905,C -2.2504,E1 24.9995,E2 -180.0809} C_DIS
Enddeposition()
LIN {X 0.3792,Y -68.8877,Z 78,A -95.0256,B 24.9048,C -2.2531,E1 25.0012,E2 -180.6748} C_DIS
Startdeposition()
$VEL.CP = VEL_PRINT
LIN {X -1.6435,Y -68.8705,Z 78,A -97.0566,B 24.9055,C -2.2442,E1 24.9955,E2 -178.6226} C_DIS
LIN {X -3.4475,Y -68.8036,Z 78,A -98.5353,B 24.9055,C -2.2446,E1 24.9913,E2 -177.1445} C_DIS
LIN {X -5.8772,Y -68.639,Z 78,A -100.6059,B 24.9055,C -2.2435,E1 24.9856,E2 -175.0705} C_DIS
LIN {X -8.3924,Y -68.377,Z 78,A -102.6709,B 24.9055,C -2.2447,E1 24.9798,E2 -173.007} C_DIS
LIN {X -10.1553,Y -68.1374,Z 78,A -104.4421,B 24.906,C -2.2381,E1 24.9749,E2 -171.2185} C_DIS
LIN {X -12.6245,Y -67.7236,Z 78,A -106.2638,B 24.9055,C -2.245,E1 24.9699,E2 -169.4114} C_DIS
LIN {X -14.3242,Y -67.3843,Z 78,A -107.9655,B 24.9059,C -2.2394,E1 24.9652,E2 -167.6944} C_DIS
LIN {X -16.7444,Y -66.8244,Z 78,A -109.776,B 24.9053,C -2.2465,E1 24.9603,E2 -165.8983} C_DIS
LIN {X -19.1429,Y -66.177,Z 78,A -111.8938,B 24.9053,C -2.2465,E1 24.9546,E2 -163.7774} C_DIS
LIN {X -21.6575,Y -65.3972,Z 78,A -114.3059,B 24.9056,C -2.243,E1 24.9482,E2 -161.3525} C_DIS
LIN {X -24.0611,Y -64.5515,Z 78,A -116.4211,B 24.9055,C -2.245,E1 24.9426,E2 -159.2377} C_DIS
LIN {X -26.3826,Y -63.6382,Z 78,A -118.2399,B 24.9048,C -2.2529,E1 24.938,E2 -157.4338} C_DIS
LIN {X -28.6577,Y -62.6465,Z 78,A -120.3203,B 24.9046,C -2.2548,E1 24.9327,E2 -155.3528} C_DIS
LIN {X -30.2655,Y -61.8857,Z 78,A -122.0534,B 24.905,C -2.2507,E1 24.9283,E2 -153.6055} C_DIS
LIN {X -32.5169,Y -60.7329,Z 78,A -123.8687,B 24.9042,C -2.2599,E1 24.9238,E2 -151.8072} C_DIS
LIN {X -34.0536,Y -59.8845,Z 78,A -125.6282,B 24.9046,C -2.2551,E1 24.9195,E2 -150.0311} C_DIS
LIN {X -36.8364,Y -58.2146,Z 78,A -128.2216,B 24.9041,C -2.2615,E1 24.9133,E2 -147.4448} C_DIS
LIN {X -38.9716,Y -56.8075,Z 78,A -130.4985,B 24.9041,C -2.2615,E1 24.9081,E2 -145.1603} C_DIS
LIN {X -41.0448,Y -55.3281,Z 78,A -132.5309,B 24.9036,C -2.267,E1 24.9035,E2 -143.1338} C_DIS
LIN {X -43.0681,Y -53.768,Z 78,A -134.6519,B 24.9033,C -2.2708,E1 24.8988,E2 -141.0142} C_DIS
LIN {X -45.0603,Y -52.1094,Z 78,A -136.8991,B 24.9031,C -2.2729,E1 24.894,E2 -138.7632} C_DIS
LIN {X -47.2303,Y -50.1498,Z 78,A -139.165,B 24.9024,C -2.2814,E1 24.8894,E2 -136.5084} C_DIS
LIN {X -49.2955,Y -48.1229,Z 78,A -141.6954,B 24.9022,C -2.2837,E1 24.8844,E2 -133.9727} C_DIS
LIN {X -51.3285,Y -45.9465,Z 78,A -144.0667,B 24.9015,C -2.2914,E1 24.8799,E2 -131.6094} C_DIS
LIN {X -52.9996,Y -44.0085,Z 78,A -146.4073,B 24.9015,C -2.2916,E1 24.8757,E2 -129.2586} C_DIS
LIN {X -54.856,Y -41.6732,Z 78,A -148.6085,B 24.9004,C -2.3035,E1 24.872,E2 -127.0754} C_DIS
LIN {X -56.3372,Y -39.6482,Z 78,A -150.7153,B 24.9,C -2.3082,E1 24.8685,E2 -124.9694} C_DIS
LIN {X -57.751,Y -37.5591,Z 78,A -152.8265,B 24.8996,C -2.3132,E1 24.8652,E2 -122.8597} C_DIS
LIN {X -59.064,Y -35.4581,Z 78,A -154.8693,B 24.8991,C -2.3189,E1 24.8623,E2 -120.82} C_DIS
LIN {X -60.323,Y -33.271,Z 78,A -156.9865,B 24.8987,C -2.324,E1 24.8593,E2 -118.7041} C_DIS
LIN {X -61.4065,Y -31.2244,Z 78,A -158.9728,B 24.8983,C -2.328,E1 24.8568,E2 -116.7165} C_DIS
LIN {X -62.2755,Y -29.4557,Z 78,A -160.6977,B 24.8981,C -2.3307,E1 24.8547,E2 -114.9887} C_DIS
LIN {X -63.3447,Y -27.079,Z 78,A -163.0513,B 24.8979,C -2.3329,E1 24.852,E2 -112.6274} C_DIS
LIN {X -64.56,Y -24.0387,Z 78,A -165.5284,B 24.8967,C -2.3459,E1 24.8495,E2 -110.1675} C_DIS
LIN {X -65.3979,Y -21.6554,Z 78,A -167.6057,B 24.8962,C -2.3525,E1 24.8476,E2 -108.0942} C_DIS
LIN {X -66.0719,Y -19.4991,Z 78,A -169.6557,B 24.896,C -2.3545,E1 24.846,E2 -106.0372} C_DIS
LIN {X -66.8328,Y -16.7102,Z 78,A -171.9285,B 24.8951,C -2.3645,E1 24.8444,E2 -103.775} C_DIS
LIN {X -67.3859,Y -14.317,Z 78,A -174.0072,B 24.8946,C -2.3699,E1 24.8431,E2 -101.6971} C_DIS
LIN {X -67.8689,Y -11.8176,Z 78,A -176.3452,B 24.8944,C -2.3719,E1 24.8419,E2 -99.3498} C_DIS
LIN {X -68.2638,Y -9.2696,Z 78,A -178.2991,B 24.8935,C -2.3825,E1 24.8411,E2 -97.4096} C_DIS
LIN {X -68.5535,Y -6.801,Z 78,A 179.6185,B 24.8929,C -2.3886,E1 24.8405,E2 -95.3295} C_DIS
LIN {X -68.7571,Y -4.2772,Z 78,A 177.3727,B 24.8926,C -2.3923,E1 24.84,E2 -93.079} C_DIS
LIN {X -68.8705,Y -1.641,Z 78,A 175.0191,B 24.8923,C -2.396,E1 24.8398,E2 -90.72} C_DIS
LIN {X -68.8705,Y 1.6423,Z 78,A 172.569,B 24.891,C -2.4104,E1 24.8398,E2 -88.2897} C_DIS
LIN {X -68.805,Y 3.4223,Z 78,A 170.77,B 24.8911,C -2.4086,E1 24.8401,E2 -86.4754} C_DIS
LIN {X -68.6369,Y 5.9034,Z 78,A 168.9668,B 24.89,C -2.4206,E1 24.8405,E2 -84.6901} C_DIS
LIN {X -68.3771,Y 8.3915,Z 78,A 166.8957,B 24.8894,C -2.4274,E1 24.8411,E2 -82.6228} C_DIS
LIN {X -68.1373,Y 10.1563,Z 78,A 165.1111,B 24.8896,C -2.4258,E1 24.8418,E2 -80.8238} C_DIS
LIN {X -67.5225,Y 13.6548,Z 78,A 162.1714,B 24.8887,C -2.4355,E1 24.8433,E2 -77.8897} C_DIS
LIN {X -66.8252,Y 16.7412,Z 78,A 159.7269,B 24.8876,C -2.4475,E1 24.8449,E2 -75.4598} C_DIS
LIN {X -66.1622,Y 19.1947,Z 78,A 157.3351,B 24.8875,C -2.4484,E1 24.8467,E2 -73.056} C_DIS
LIN {X -65.3945,Y 21.6655,Z 78,A 155.1933,B 24.8869,C -2.4552,E1 24.8485,E2 -70.9183} C_DIS
LIN {X -64.5547,Y 24.0526,Z 78,A 153.0718,B 24.8863,C -2.4612,E1 24.8505,E2 -68.7993} C_DIS
LIN {X -63.6457,Y 26.3649,Z 78,A 151.2526,B 24.8853,C -2.4726,E1 24.8524,E2 -66.997} C_DIS
LIN {X -62.6481,Y 28.6542,Z 78,A 149.1272,B 24.8848,C -2.4778,E1 24.8548,E2 -64.8723} C_DIS
LIN {X -61.5197,Y 31.0029,Z 78,A 146.9842,B 24.8841,C -2.4846,E1 24.8575,E2 -62.7341} C_DIS
LIN {X -60.3451,Y 33.2315,Z 78,A 144.8738,B 24.8836,C -2.4904,E1 24.8602,E2 -60.6262} C_DIS
LIN {X -59.0884,Y 35.418,Z 78,A 142.4704,B 24.8836,C -2.4899,E1 24.8637,E2 -58.2093} C_DIS
LIN {X -57.7524,Y 37.557,Z 78,A 140.3596,B 24.8831,C -2.4954,E1 24.8668,E2 -56.101} C_DIS
LIN {X -56.34,Y 39.6442,Z 78,A 138.2519,B 24.8826,C -2.5009,E1 24.8702,E2 -53.9959} C_DIS
LIN {X -54.5821,Y 42.0297,Z 78,A 135.7793,B 24.882,C -2.5073,E1 24.8743,E2 -51.5266} C_DIS
LIN {X -52.703,Y 44.3651,Z 78,A 133.369,B 24.8812,C -2.5154,E1 24.8786,E2 -49.1246} C_DIS
LIN {X -51.0241,Y 46.286,Z 78,A 131.2385,B 24.8807,C -2.5205,E1 24.8825,E2 -46.9968} C_DIS
LIN {X -49.2911,Y 48.1274,Z 78,A 129.1296,B 24.8803,C -2.5255,E1 24.8866,E2 -44.8907} C_DIS
LIN {X -47.5086,Y 49.8879,Z 78,A 127.0226,B 24.8799,C -2.5299,E1 24.8908,E2 -42.7854} C_DIS
LIN {X -45.4048,Y 51.8085,Z 78,A 124.602,B 24.8795,C -2.5341,E1 24.8959,E2 -40.3652} C_DIS
LIN {X -42.9753,Y 53.8417,Z 78,A 121.8978,B 24.8791,C -2.5383,E1 24.9017,E2 -37.6608} C_DIS
LIN {X -40.9643,Y 55.3871,Z 78,A 119.7971,B 24.8786,C -2.5428,E1 24.9064,E2 -35.5634} C_DIS
LIN {X -38.9213,Y 56.8415,Z 78,A 117.7007,B 24.8782,C -2.5467,E1 24.9112,E2 -33.4691} C_DIS
LIN {X -36.5132,Y 58.4165,Z 78,A 115.4311,B 24.8776,C -2.5539,E1 24.9165,E2 -31.2093} C_DIS
LIN {X -33.9828,Y 59.9251,Z 78,A 113.1241,B 24.8768,C -2.5614,E1 24.9221,E2 -28.9132} C_DIS
LIN {X -31.7607,Y 61.1319,Z 78,A 111.018,B 24.8765,C -2.5648,E1 24.9272,E2 -26.8094} C_DIS
LIN {X -29.7709,Y 62.124,Z 78,A 109.0546,B 24.8765,C -2.5652,E1 24.9322,E2 -24.8418} C_DIS
LIN {X -27.1895,Y 63.2975,Z 78,A 106.7995,B 24.8759,C -2.5709,E1 24.9379,E2 -22.595} C_DIS
LIN {X -25.5459,Y 63.9785,Z 78,A 105.008,B 24.8764,C -2.566,E1 24.9426,E2 -20.7877} C_DIS
LIN {X -22.8362,Y 64.9939,Z 78,A 102.627,B 24.876,C -2.5696,E1 24.9488,E2 -18.4106} C_DIS
LIN {X -19.9812,Y 65.9289,Z 78,A 100.3657,B 24.8752,C -2.5778,E1 24.9548,E2 -16.1648} C_DIS
LIN {X -17.592,Y 66.6061,Z 78,A 98.286,B 24.8751,C -2.5796,E1 24.9604,E2 -14.0861} C_DIS
LIN {X -15.8656,Y 67.0382,Z 78,A 96.5512,B 24.8755,C -2.5752,E1 24.9651,E2 -12.3384} C_DIS
LIN {X -13.3928,Y 67.5757,Z 78,A 94.4403,B 24.8753,C -2.5768,E1 24.9709,E2 -10.2288} C_DIS
LIN {X -10.2882,Y 68.1169,Z 78,A 92.0811,B 24.8746,C -2.5847,E1 24.9774,E2 -7.8862} C_DIS
LIN {X -8.3715,Y 68.3794,Z 78,A 90.2042,B 24.8751,C -2.5794,E1 24.9826,E2 -5.9954} C_DIS
LIN {X -5.8549,Y 68.6408,Z 78,A 88.0999,B 24.875,C -2.5804,E1 24.9884,E2 -3.8925} C_DIS
LIN {X -3.3298,Y 68.8095,Z 78,A 85.9914,B 24.875,C -2.5811,E1 24.9943,E2 -1.785} C_DIS
LIN {X -0.3173,Y 68.8884,Z 78,A 83.6972,B 24.8744,C -2.5868,E1 25.0007,E2 0.496} C_DIS
LIN {X 1.7514,Y 68.8677,Z 78,A 81.7661,B 24.8748,C -2.582,E1 25.0061,E2 2.4381} C_DIS
Enddeposition()
END
